KUKA KRL program: MyProgram_244().src

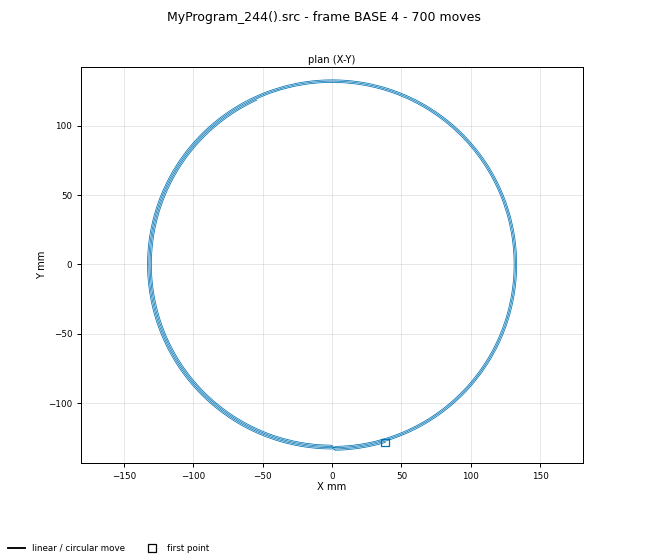
[picture p0: tool path of MyProgram_244().src in frame BASE 4, 700 of 700 moves have a stored position in this frame; points joined in program order, loops and branches not executed]
&ACCESS RVP
&REL 1
&PARAM TEMPLATE = C:\KRC\Roboter\Template\vorgabe
&PARAM EDITMASK = *
DEF MyProgram_244()
; ---- Setting reference (Base) ----
$BASE = BASE_DATA[4]

; --------------------------
; ---- Setting tool (TCP) ----
$TOOL = TOOL_DATA[3]
; --------------------------

$VEL.CP = VEL_APROX_PRINT
Startdeposition()
$VEL.CP = VEL_PRINT
LIN {X 38.4401,Y -128.4466,Z 162,A -74.7058,B 18.9491,C -0.3329,E1 18.9974,E2 523.2154} C_DIS
LIN {X 33.1101,Y -129.9203,Z 162,A -77.04,B 18.9491,C -0.3317,E1 18.9911,E2 525.548} C_DIS
LIN {X 29.9609,Y -130.6824,Z 162,A -78.4866,B 18.9492,C -0.328,E1 18.9871,E2 527.0033} C_DIS
LIN {X 25.973,Y -131.5353,Z 162,A -80.3087,B 18.9492,C -0.3233,E1 18.9821,E2 528.8368} C_DIS
LIN {X 22.2371,Y -132.2161,Z 162,A -81.8211,B 18.9492,C -0.3266,E1 18.978,E2 530.3367} C_DIS
LIN {X 19.1741,Y -132.6951,Z 162,A -83.027,B 18.9492,C -0.3306,E1 18.9747,E2 531.5289} C_DIS
LIN {X 16.3892,Y -133.0686,Z 162,A -84.4176,B 18.9493,C -0.3222,E1 18.9708,E2 532.9437} C_DIS
LIN {X 12.9583,Y -133.4455,Z 162,A -85.833,B 18.9493,C -0.3239,E1 18.9668,E2 534.3526} C_DIS
LIN {X 9.2967,Y -133.7512,Z 162,A -87.5113,B 18.9493,C -0.3189,E1 18.9621,E2 536.0452} C_DIS
LIN {X 5.2547,Y -133.9702,Z 162,A -89.0028,B 18.9493,C -0.3279,E1 18.9581,E2 537.5084} C_DIS
LIN {X 2.1511,Y -134.056,Z 162,A -90.4324,B 18.9493,C -0.3234,E1 18.954,E2 538.9513} C_DIS
LIN {X 2.1511,Y -134.056,Z 162,A -90.4324,B 18.9493,C -0.3234,E1 18.954,E2 538.9513} C_DIS
Enddeposition()
LIN {X 0.9211,Y -133.1439,Z 162,A -90.13,B 17.7288,C -0.2117,E1 17.7322,E2 538.9153} C_DIS
Startdeposition()
$VEL.CP = VEL_PRINT
LIN {X 4.405,Y -133.0795,Z 162,A -88.3392,B 17.7287,C -0.2229,E1 17.7373,E2 537.088} C_DIS
LIN {X 8.2716,Y -132.8933,Z 162,A -86.7196,B 17.7287,C -0.2218,E1 17.7418,E2 535.4731} C_DIS
LIN {X 12.4751,Y -132.5649,Z 162,A -84.9551,B 17.7287,C -0.2207,E1 17.7467,E2 533.7136} C_DIS
LIN {X 16.1435,Y -132.1686,Z 162,A -83.269,B 17.7287,C -0.2253,E1 17.7514,E2 532.0144} C_DIS
LIN {X 20.3858,Y -131.5804,Z 162,A -81.5673,B 17.7287,C -0.221,E1 17.756,E2 530.3288} C_DIS
LIN {X 23.9672,Y -130.9764,Z 162,A -79.9126,B 17.7287,C -0.2256,E1 17.7606,E2 528.6617} C_DIS
LIN {X 28.0553,Y -130.1609,Z 162,A -78.17,B 17.7287,C -0.2251,E1 17.7654,E2 526.924} C_DIS
LIN {X 32.1027,Y -129.2239,Z 162,A -76.0026,B 17.7285,C -0.2413,E1 17.7714,E2 524.7081} C_DIS
LIN {X 35.7552,Y -128.2596,Z 162,A -74.7161,B 17.7286,C -0.2299,E1 17.7747,E2 523.4623} C_DIS
LIN {X 38.9324,Y -127.3311,Z 162,A -72.9424,B 17.7284,C -0.2449,E1 17.7796,E2 521.6439} C_DIS
LIN {X 42.8761,Y -126.0602,Z 162,A -71.6301,B 17.7286,C -0.2287,E1 17.7829,E2 520.3885} C_DIS
LIN {X 46.937,Y -124.603,Z 162,A -69.7312,B 17.7286,C -0.2326,E1 17.7879,E2 518.4825} C_DIS
LIN {X 49.968,Y -123.4186,Z 162,A -68.3823,B 17.7286,C -0.2324,E1 17.7914,E2 517.1386} C_DIS
LIN {X 52.8742,Y -122.2016,Z 162,A -67.036,B 17.7286,C -0.2339,E1 17.7949,E2 515.7921} C_DIS
LIN {X 55.7231,Y -120.9292,Z 162,A -65.1103,B 17.7282,C -0.2587,E1 17.8,E2 513.7926} C_DIS
LIN {X 59.9495,Y -118.8916,Z 162,A -63.7898,B 17.7285,C -0.2344,E1 17.803,E2 512.5568} C_DIS
LIN {X 62.5044,Y -117.5693,Z 162,A -61.9097,B 17.7282,C -0.2615,E1 17.8079,E2 510.5957} C_DIS
LIN {X 66.4149,Y -115.4063,Z 162,A -60.4001,B 17.7284,C -0.2485,E1 17.8114,E2 509.1353} C_DIS
LIN {X 70.1912,Y -113.1488,Z 162,A -58.4889,B 17.7284,C -0.2525,E1 17.816,E2 507.2197} C_DIS
LIN {X 76.278,Y -109.1383,Z 162,A -55.6866,B 17.7284,C -0.2452,E1 17.8224,E2 504.4551} C_DIS
LIN {X 78.609,Y -107.4715,Z 162,A -53.6651,B 17.7279,C -0.2788,E1 17.8272,E2 502.3342} C_DIS
LIN {X 82.5719,Y -104.458,Z 162,A -51.8372,B 17.728,C -0.2706,E1 17.8311,E2 500.5428} C_DIS
LIN {X 85.1779,Y -102.3438,Z 162,A -50.6123,B 17.7281,C -0.265,E1 17.8337,E2 499.3433} C_DIS
LIN {X 88.5691,Y -99.4237,Z 162,A -48.703,B 17.7281,C -0.2685,E1 17.8377,E2 497.4335} C_DIS
LIN {X 92.9776,Y -95.3137,Z 162,A -45.9022,B 17.7279,C -0.2826,E1 17.8434,E2 494.6036} C_DIS
LIN {X 95.4007,Y -92.8885,Z 162,A -44.7083,B 17.7279,C -0.2748,E1 17.8457,E2 493.4425} C_DIS
LIN {X 98.1153,Y -90.0157,Z 162,A -43.0038,B 17.7279,C -0.279,E1 17.8489,E2 491.7353} C_DIS
LIN {X 102.4796,Y -85.0139,Z 162,A -40.1393,B 17.7279,C -0.2863,E1 17.8542,E2 488.8659} C_DIS
LIN {X 107.576,Y -78.4665,Z 162,A -36.8646,B 17.7279,C -0.2835,E1 17.8597,E2 485.6228} C_DIS
LIN {X 112.5667,Y -71.1208,Z 162,A -33.2021,B 17.7278,C -0.2872,E1 17.8654,E2 481.9748} C_DIS
LIN {X 115.0297,Y -67.0654,Z 162,A -30.8023,B 17.7275,C -0.3071,E1 17.8689,E2 479.5279} C_DIS
LIN {X 118.2387,Y -61.2296,Z 162,A -27.4523,B 17.727,C -0.3348,E1 17.8734,E2 476.1134} C_DIS
LIN {X 120.3127,Y -57.043,Z 162,A -26.0674,B 17.7273,C -0.3152,E1 17.875,E2 474.8032} C_DIS
LIN {X 121.6559,Y -54.1186,Z 162,A -24.6633,B 17.7273,C -0.3199,E1 17.8766,E2 473.3947} C_DIS
LIN {X 123.1449,Y -50.6435,Z 162,A -23.0597,B 17.7272,C -0.3237,E1 17.8783,E2 471.7916} C_DIS
LIN {X 125.0396,Y -45.7649,Z 162,A -20.8991,B 17.7272,C -0.3267,E1 17.8805,E2 469.639} C_DIS
LIN {X 126.4553,Y -41.691,Z 162,A -18.9776,B 17.727,C -0.3348,E1 17.8822,E2 467.7065} C_DIS
LIN {X 127.8269,Y -37.2725,Z 162,A -17.0387,B 17.727,C -0.3387,E1 17.8838,E2 465.7711} C_DIS
LIN {X 128.7106,Y -34.0968,Z 162,A -15.5705,B 17.7268,C -0.345,E1 17.8848,E2 464.2947} C_DIS
LIN {X 129.7402,Y -29.942,Z 162,A -13.3916,B 17.7264,C -0.3643,E1 17.8863,E2 462.0712} C_DIS
LIN {X 130.5248,Y -26.3116,Z 162,A -12.4598,B 17.7268,C -0.3422,E1 17.8868,E2 461.2194} C_DIS
LIN {X 130.9612,Y -24.052,Z 162,A -11.1753,B 17.7266,C -0.3571,E1 17.8874,E2 459.8973} C_DIS
LIN {X 131.4541,Y -21.1975,Z 162,A -9.8457,B 17.7264,C -0.3643,E1 17.888,E2 458.5556} C_DIS
LIN {X 132.0314,Y -17.2257,Z 162,A -8.2288,B 17.7264,C -0.3652,E1 17.8887,E2 456.9497} C_DIS
LIN {X 132.4714,Y -13.4488,Z 162,A -6.5412,B 17.7263,C -0.3723,E1 17.8892,E2 455.2535} C_DIS
LIN {X 132.801,Y -9.6401,Z 162,A -5.0073,B 17.7263,C -0.3729,E1 17.8895,E2 453.7309} C_DIS
LIN {X 133.0236,Y -5.8476,Z 162,A -3.2243,B 17.726,C -0.384,E1 17.8897,E2 451.9273} C_DIS
LIN {X 133.1445,Y -1.4544,Z 162,A -1.4344,B 17.726,C -0.3857,E1 17.8898,E2 450.1472} C_DIS
LIN {X 133.1283,Y 2.4386,Z 162,A 0.2134,B 17.7259,C -0.3898,E1 17.8898,E2 448.5003} C_DIS
LIN {X 132.9874,Y 6.5875,Z 162,A 1.9267,B 17.7259,C -0.3923,E1 17.8896,E2 446.7935} C_DIS
LIN {X 132.7248,Y 10.6513,Z 162,A 3.744,B 17.7257,C -0.4003,E1 17.8892,E2 444.9659} C_DIS
LIN {X 132.3728,Y 14.3688,Z 162,A 5.2397,B 17.7257,C -0.4008,E1 17.8888,E2 443.4817} C_DIS
LIN {X 131.8824,Y 18.338,Z 162,A 7.0014,B 17.7255,C -0.4077,E1 17.8882,E2 441.7126} C_DIS
LIN {X 131.2981,Y 22.1322,Z 162,A 8.5557,B 17.7255,C -0.4087,E1 17.8875,E2 440.1681} C_DIS
LIN {X 130.6424,Y 25.7311,Z 162,A 11.1257,B 17.7244,C -0.4538,E1 17.886,E2 437.473} C_DIS
LIN {X 129.1593,Y 32.3575,Z 162,A 12.8777,B 17.7253,C -0.4151,E1 17.885,E2 435.8619} C_DIS
LIN {X 128.1707,Y 36.0732,Z 162,A 14.7264,B 17.7251,C -0.4278,E1 17.8836,E2 433.9874} C_DIS
LIN {X 125.561,Y 44.3161,Z 162,A 18.3458,B 17.7249,C -0.4344,E1 17.8805,E2 430.3762} C_DIS
LIN {X 124.6316,Y 46.8606,Z 162,A 19.568,B 17.7248,C -0.44,E1 17.8793,E2 429.1457} C_DIS
LIN {X 123.1266,Y 50.6874,Z 162,A 21.3856,B 17.7246,C -0.4469,E1 17.8774,E2 427.3203} C_DIS
LIN {X 121.6302,Y 54.176,Z 162,A 22.9095,B 17.7246,C -0.4471,E1 17.8757,E2 425.8079} C_DIS
LIN {X 119.6437,Y 58.432,Z 162,A 25.2502,B 17.7241,C -0.4654,E1 17.8728,E2 423.4259} C_DIS
LIN {X 118.0607,Y 61.5686,Z 162,A 26.232,B 17.7246,C -0.4483,E1 17.8716,E2 422.5074} C_DIS
LIN {X 116.6222,Y 64.2555,Z 162,A 27.8267,B 17.7242,C -0.463,E1 17.8694,E2 420.877} C_DIS
LIN {X 114.3351,Y 68.2415,Z 162,A 29.7403,B 17.7242,C -0.4656,E1 17.8668,E2 418.9691} C_DIS
LIN {X 111.9815,Y 72.0392,Z 162,A 31.6763,B 17.724,C -0.471,E1 17.8639,E2 417.0298} C_DIS
LIN {X 109.5783,Y 75.6449,Z 162,A 33.5648,B 17.7238,C -0.4766,E1 17.8609,E2 415.1367} C_DIS
LIN {X 106.6136,Y 79.7687,Z 162,A 35.6684,B 17.7238,C -0.4786,E1 17.8574,E2 413.0413} C_DIS
LIN {X 104.0275,Y 83.113,Z 162,A 37.4895,B 17.7237,C -0.483,E1 17.8543,E2 411.2185} C_DIS
LIN {X 101.2433,Y 86.4831,Z 162,A 39.3875,B 17.7235,C -0.4879,E1 17.8509,E2 409.3169} C_DIS
LIN {X 98.3103,Y 89.8036,Z 162,A 41.3124,B 17.7235,C -0.4928,E1 17.8473,E2 407.3884} C_DIS
LIN {X 95.1732,Y 93.1209,Z 162,A 43.2319,B 17.7233,C -0.4953,E1 17.8436,E2 405.4731} C_DIS
LIN {X 91.8689,Y 96.3823,Z 162,A 45.2066,B 17.7233,C -0.4985,E1 17.8396,E2 403.4999} C_DIS
LIN {X 88.5887,Y 99.4061,Z 162,A 47.1354,B 17.7231,C -0.5026,E1 17.8356,E2 401.5688} C_DIS
LIN {X 85.7795,Y 101.8399,Z 162,A 48.7338,B 17.7231,C -0.5056,E1 17.8322,E2 399.9698} C_DIS
LIN {X 82.2394,Y 104.7192,Z 162,A 50.6526,B 17.7231,C -0.5075,E1 17.828,E2 398.0553} C_DIS
LIN {X 78.5721,Y 107.4986,Z 162,A 52.6154,B 17.7229,C -0.5103,E1 17.8236,E2 396.0938} C_DIS
LIN {X 74.9854,Y 110.0308,Z 162,A 54.6052,B 17.7227,C -0.5173,E1 17.819,E2 394.091} C_DIS
LIN {X 71.1647,Y 112.5389,Z 162,A 56.4761,B 17.7227,C -0.5166,E1 17.8147,E2 392.231} C_DIS
LIN {X 66.9137,Y 115.1174,Z 162,A 58.7367,B 17.7225,C -0.5244,E1 17.8092,E2 389.9551} C_DIS
LIN {X 63.2973,Y 117.1451,Z 162,A 60.3738,B 17.7226,C -0.5212,E1 17.8052,E2 388.3354} C_DIS
LIN {X 59.7268,Y 119.0044,Z 162,A 61.9869,B 17.7226,C -0.519,E1 17.8013,E2 386.7363} C_DIS
LIN {X 56.9965,Y 120.3349,Z 162,A 63.3153,B 17.7226,C -0.5214,E1 17.7979,E2 385.4051} C_DIS
LIN {X 54.0101,Y 121.7044,Z 162,A 64.8105,B 17.7225,C -0.5261,E1 17.7941,E2 383.8998} C_DIS
LIN {X 49.8646,Y 123.4603,Z 162,A 66.6914,B 17.7225,C -0.5261,E1 17.7892,E2 382.0255} C_DIS
LIN {X 46.3817,Y 124.811,Z 162,A 68.2314,B 17.7225,C -0.5251,E1 17.7852,E2 380.4936} C_DIS
LIN {X 43.3739,Y 125.8876,Z 162,A 69.6353,B 17.7225,C -0.5274,E1 17.7815,E2 379.0862} C_DIS
LIN {X 40.0822,Y 126.9747,Z 162,A 71.3845,B 17.7221,C -0.5383,E1 17.7768,E2 377.306} C_DIS
LIN {X 35.6883,Y 128.2783,Z 162,A 73.0222,B 17.7225,C -0.5272,E1 17.7725,E2 375.7088} C_DIS
LIN {X 32.7382,Y 129.0626,Z 162,A 75.134,B 17.7215,C -0.558,E1 17.7666,E2 373.5005} C_DIS
LIN {X 27.2206,Y 130.3399,Z 162,A 76.7611,B 17.7224,C -0.5289,E1 17.7624,E2 371.972} C_DIS
LIN {X 23.9894,Y 130.9724,Z 162,A 78.318,B 17.7222,C -0.5348,E1 17.758,E2 370.3985} C_DIS
LIN {X 20.4151,Y 131.5759,Z 162,A 79.8044,B 17.7223,C -0.5326,E1 17.754,E2 368.9214} C_DIS
LIN {X 16.969,Y 132.065,Z 162,A 81.3445,B 17.7223,C -0.5346,E1 17.7497,E2 367.3765} C_DIS
LIN {X 12.8514,Y 132.5288,Z 162,A 83.0922,B 17.7223,C -0.5337,E1 17.7449,E2 365.6337} C_DIS
LIN {X 8.8949,Y 132.8549,Z 162,A 84.9027,B 17.7222,C -0.5376,E1 17.7398,E2 363.8117} C_DIS
LIN {X 4.989,Y 133.0571,Z 162,A 86.4461,B 17.7223,C -0.5325,E1 17.7355,E2 362.2857} C_DIS
LIN {X 0.9974,Y 133.147,Z 162,A 88.2211,B 17.7223,C -0.5345,E1 17.7305,E2 360.5046} C_DIS
LIN {X -2.4674,Y 133.1279,Z 162,A 89.7391,B 17.7223,C -0.5352,E1 17.7263,E2 358.9841} C_DIS
LIN {X -6.5137,Y 132.9911,Z 162,A 91.4349,B 17.7223,C -0.5331,E1 17.7216,E2 357.2948} C_DIS
LIN {X -9.9735,Y 132.7766,Z 162,A 92.9352,B 17.7223,C -0.5329,E1 17.7174,E2 355.7943} C_DIS
LIN {X -14.1183,Y 132.3998,Z 162,A 94.7247,B 17.7223,C -0.5321,E1 17.7124,E2 354.0061} C_DIS
LIN {X -17.8365,Y 131.9513,Z 162,A 96.4127,B 17.7223,C -0.534,E1 17.7077,E2 352.3101} C_DIS
LIN {X -21.7102,Y 131.3685,Z 162,A 98.327,B 17.722,C -0.5413,E1 17.7024,E2 350.3695} C_DIS
LIN {X -24.9922,Y 130.7837,Z 162,A 99.4282,B 17.7224,C -0.5283,E1 17.6995,E2 349.3093} C_DIS
LIN {X -31.9254,Y 129.2683,Z 162,A 102.4778,B 17.7225,C -0.5256,E1 17.6912,E2 346.2628} C_DIS
LIN {X -34.6255,Y 128.5696,Z 162,A 103.794,B 17.7225,C -0.5287,E1 17.6876,E2 344.9337} C_DIS
LIN {X -43.6563,Y 125.7897,Z 162,A 107.4467,B 17.723,C -0.5097,E1 17.678,E2 341.334} C_DIS
LIN {X -46.9349,Y 124.6038,Z 162,A 109.308,B 17.7226,C -0.5207,E1 17.673,E2 339.4312} C_DIS
LIN {X -50.5818,Y 123.1707,Z 162,A 111.3581,B 17.7223,C -0.5314,E1 17.6676,E2 337.3393} C_DIS
LIN {X -53.8283,Y 121.7857,Z 162,A 112.4133,B 17.7229,C -0.513,E1 17.6651,E2 336.3411} C_DIS
LIN {X -56.6826,Y 120.4849,Z 162,A 114.1908,B 17.7225,C -0.5261,E1 17.6604,E2 334.5138} C_DIS
LIN {X -59.6374,Y 119.0489,Z 162,A 115.973,B 17.7222,C -0.537,E1 17.6559,E2 332.6888} C_DIS
LIN {X -64.3129,Y 116.5904,Z 162,A 117.425,B 17.7231,C -0.5046,E1 17.6526,E2 331.3378} C_DIS
LIN {X -66.9437,Y 115.1001,Z 162,A 118.9992,B 17.7229,C -0.512,E1 17.6487,E2 329.7325} C_DIS
LIN {X -70.7861,Y 112.7779,Z 162,A 121.021,B 17.7229,C -0.5117,E1 17.6438,E2 327.7021} C_DIS
LIN {X -74.994,Y 110.025,Z 162,A 123.0696,B 17.7231,C -0.5038,E1 17.6391,E2 325.6699} C_DIS
LIN {X -79.5511,Y 106.7756,Z 162,A 125.2577,B 17.7234,C -0.4916,E1 17.6343,E2 323.5109} C_DIS
LIN {X -82.004,Y 104.904,Z 162,A 126.8766,B 17.7232,C -0.499,E1 17.6306,E2 321.859} C_DIS
LIN {X -85.898,Y 101.739,Z 162,A 129.4235,B 17.723,C -0.5079,E1 17.625,E2 319.2684} C_DIS
LIN {X -89.1638,Y 98.8909,Z 162,A 130.7262,B 17.7236,C -0.4845,E1 17.6225,E2 318.0354} C_DIS
LIN {X -91.6865,Y 96.5567,Z 162,A 132.9844,B 17.723,C -0.5081,E1 17.6177,E2 315.6857} C_DIS
LIN {X -95.4305,Y 92.8577,Z 162,A 135.1689,B 17.7232,C -0.5001,E1 17.6135,E2 313.5139} C_DIS
LIN {X -98.6883,Y 89.3871,Z 162,A 136.5035,B 17.724,C -0.4708,E1 17.6111,E2 312.2677} C_DIS
LIN {X -100.9612,Y 86.8116,Z 162,A 138.3748,B 17.7237,C -0.4807,E1 17.6076,E2 310.3515} C_DIS
LIN {X -104.1069,Y 83.0131,Z 162,A 140.3623,B 17.724,C -0.4708,E1 17.6042,E2 308.3832} C_DIS
LIN {X -106.758,Y 79.5748,Z 162,A 142.2426,B 17.7241,C -0.4665,E1 17.601,E2 306.504} C_DIS
LIN {X -109.469,Y 75.8026,Z 162,A 144.4981,B 17.7241,C -0.47,E1 17.5973,E2 304.2206} C_DIS
LIN {X -111.4017,Y 72.9328,Z 162,A 145.6418,B 17.7244,C -0.4543,E1 17.5956,E2 303.1204} C_DIS
LIN {X -114.2198,Y 68.4351,Z 162,A 147.7787,B 17.7247,C -0.4432,E1 17.5925,E2 301.0043} C_DIS
LIN {X -115.7253,Y 65.8566,Z 162,A 149.3559,B 17.7245,C -0.4495,E1 17.5903,E2 299.3942} C_DIS
LIN {X -117.7258,Y 62.2065,Z 162,A 151.5968,B 17.7243,C -0.4598,E1 17.5873,E2 297.1018} C_DIS
LIN {X -119.7405,Y 58.234,Z 162,A 153.2256,B 17.7246,C -0.4446,E1 17.5853,E2 295.5106} C_DIS
LIN {X -121.8148,Y 53.7632,Z 162,A 155.3479,B 17.7248,C -0.4386,E1 17.5829,E2 293.3912} C_DIS
LIN {X -124.1451,Y 48.1345,Z 162,A 157.7942,B 17.7251,C -0.425,E1 17.5804,E2 290.9698} C_DIS
LIN {X -125.3038,Y 45.0323,Z 162,A 159.2043,B 17.7252,C -0.4203,E1 17.579,E2 289.5636} C_DIS
LIN {X -126.5386,Y 41.4408,Z 162,A 161.1164,B 17.7252,C -0.4248,E1 17.5773,E2 287.6207} C_DIS
LIN {X -128.4223,Y 35.1736,Z 162,A 163.6718,B 17.7255,C -0.4076,E1 17.5753,E2 285.1008} C_DIS
LIN {X -129.1451,Y 32.4134,Z 162,A 164.9402,B 17.7255,C -0.4053,E1 17.5744,E2 283.8293} C_DIS
LIN {X -130.6342,Y 25.7741,Z 162,A 168.2618,B 17.7255,C -0.4095,E1 17.5725,E2 280.4649} C_DIS
LIN {X -131.2524,Y 22.4034,Z 162,A 169.5416,B 17.7257,C -0.3985,E1 17.5719,E2 279.2107} C_DIS
LIN {X -131.8734,Y 18.4007,Z 162,A 171.7432,B 17.7255,C -0.4086,E1 17.571,E2 276.9563} C_DIS
LIN {X -132.4547,Y 13.6075,Z 162,A 173.4419,B 17.7259,C -0.3894,E1 17.5705,E2 275.3064} C_DIS
LIN {X -132.7637,Y 10.1499,Z 162,A 174.8116,B 17.7261,C -0.3806,E1 17.5702,E2 273.9538} C_DIS
LIN {X -133.0072,Y 6.1945,Z 162,A 176.5855,B 17.7261,C -0.3776,E1 17.57,E2 272.1741} C_DIS
LIN {X -133.1499,Y 0.6535,Z 162,A 179.0729,B 17.7262,C -0.3737,E1 17.5698,E2 269.6778} C_DIS
LIN {X -133.0912,Y -3.9837,Z 162,A -179.0232,B 17.7264,C -0.3644,E1 17.57,E2 267.7877} C_DIS
LIN {X -132.9015,Y -8.1385,Z 162,A -177.2896,B 17.7266,C -0.3571,E1 17.5702,E2 266.0633} C_DIS
LIN {X -132.51,Y -13.0469,Z 162,A -175.2686,B 17.7268,C -0.3473,E1 17.5707,E2 264.057} C_DIS
LIN {X -131.6927,Y -19.6607,Z 162,A -172.319,B 17.7268,C -0.3412,E1 17.5718,E2 261.1016} C_DIS
LIN {X -131.0164,Y -23.7438,Z 162,A -170.2086,B 17.7268,C -0.347,E1 17.5728,E2 258.9537} C_DIS
LIN {X -130.3,Y -27.4114,Z 162,A -168.7136,B 17.7269,C -0.3383,E1 17.5736,E2 257.4746} C_DIS
LIN {X -129.2408,Y -32.0364,Z 162,A -166.8324,B 17.7271,C -0.3269,E1 17.5748,E2 255.6153} C_DIS
LIN {X -128.2073,Y -35.9422,Z 162,A -165.0386,B 17.7271,C -0.3236,E1 17.5761,E2 253.8169} C_DIS
LIN {X -127.2376,Y -39.2379,Z 162,A -163.5455,B 17.7273,C -0.3198,E1 17.5773,E2 252.3239} C_DIS
LIN {X -126.252,Y -42.3016,Z 162,A -162.1634,B 17.7273,C -0.3157,E1 17.5785,E2 250.9438} C_DIS
LIN {X -125.0828,Y -45.6452,Z 162,A -160.6097,B 17.7273,C -0.3124,E1 17.58,E2 249.3883} C_DIS
LIN {X -123.4363,Y -49.924,Z 162,A -158.6021,B 17.7275,C -0.308,E1 17.582,E2 247.3787} C_DIS
LIN {X -122.0265,Y -53.2791,Z 162,A -156.9886,B 17.7275,C -0.3053,E1 17.5838,E2 245.7612} C_DIS
LIN {X -118.9985,Y -59.7395,Z 162,A -153.9874,B 17.7277,C -0.2945,E1 17.5874,E2 242.7717} C_DIS
LIN {X -117.7216,Y -62.2144,Z 162,A -152.7089,B 17.7277,C -0.2941,E1 17.5891,E2 241.4847} C_DIS
LIN {X -115.6817,Y -65.933,Z 162,A -150.8034,B 17.7277,C -0.2921,E1 17.5917,E2 239.5714} C_DIS
LIN {X -113.3681,Y -69.8366,Z 162,A -148.659,B 17.7277,C -0.2937,E1 17.5948,E2 237.4056} C_DIS
LIN {X -110.985,Y -73.5658,Z 162,A -147.1433,B 17.728,C -0.2755,E1 17.5971,E2 235.9388} C_DIS
LIN {X -109.1237,Y -76.299,Z 162,A -145.5502,B 17.728,C -0.2779,E1 17.5996,E2 234.3263} C_DIS
LIN {X -106.6318,Y -79.7443,Z 162,A -143.6861,B 17.728,C -0.2747,E1 17.6027,E2 232.4596} C_DIS
LIN {X -103.9378,Y -83.2256,Z 162,A -141.8161,B 17.728,C -0.2695,E1 17.6059,E2 230.5941} C_DIS
LIN {X -101.4436,Y -86.2474,Z 162,A -139.679,B 17.7279,C -0.2814,E1 17.6099,E2 228.4032} C_DIS
LIN {X -98.758,Y -89.3102,Z 162,A -138.6032,B 17.7283,C -0.2539,E1 17.6117,E2 227.4112} C_DIS
LIN {X -96.7778,Y -91.4521,Z 162,A -137.0477,B 17.7282,C -0.2617,E1 17.6148,E2 225.8202} C_DIS
LIN {X -93.7145,Y -94.5888,Z 162,A -135.119,B 17.7282,C -0.2592,E1 17.6186,E2 223.8876} C_DIS
LIN {X -90.3961,Y -97.7656,Z 162,A -133.3724,B 17.7284,C -0.2472,E1 17.622,E2 222.1702} C_DIS
LIN {X -88.1061,Y -99.8336,Z 162,A -131.8304,B 17.7284,C -0.2522,E1 17.6253,E2 220.6029} C_DIS
LIN {X -83.005,Y -104.1134,Z 162,A -129.1857,B 17.7284,C -0.2391,E1 17.631,E2 217.9866} C_DIS
LIN {X -80.5913,Y -105.9934,Z 162,A -127.5502,B 17.7284,C -0.2481,E1 17.6346,E2 216.313} C_DIS
LIN {X -77.769,Y -108.0813,Z 162,A -125.9641,B 17.7284,C -0.2482,E1 17.6382,E2 214.7183} C_DIS
LIN {X -74.2414,Y -110.534,Z 162,A -124.1683,B 17.7284,C -0.2434,E1 17.6424,E2 212.9297} C_DIS
LIN {X -70.2026,Y -113.1414,Z 162,A -121.9915,B 17.7284,C -0.2441,E1 17.6475,E2 210.7404} C_DIS
LIN {X -67.1395,Y -114.9862,Z 162,A -120.5861,B 17.7285,C -0.2371,E1 17.6509,E2 209.3518} C_DIS
LIN {X -63.395,Y -117.0925,Z 162,A -118.7317,B 17.7285,C -0.2349,E1 17.6554,E2 207.4972} C_DIS
LIN {X -60.2441,Y -118.7416,Z 162,A -117.2429,B 17.7285,C -0.2315,E1 17.6591,E2 206.0137} C_DIS
LIN {X -57.0225,Y -120.3225,Z 162,A -115.621,B 17.7285,C -0.2324,E1 17.6632,E2 204.3825} C_DIS
LIN {X -52.9041,Y -122.1887,Z 162,A -113.7705,B 17.7286,C -0.2269,E1 17.6679,E2 202.5438} C_DIS
LIN {X -49.376,Y -123.6572,Z 162,A -112.1541,B 17.7286,C -0.2242,E1 17.6721,E2 200.931} C_DIS
LIN {X -46.0174,Y -124.9474,Z 162,A -110.4396,B 17.7286,C -0.2288,E1 17.6766,E2 199.1963} C_DIS
LIN {X -41.7412,Y -126.4386,Z 162,A -108.6802,B 17.7287,C -0.2203,E1 17.6812,E2 197.4601} C_DIS
LIN {X -38.8691,Y -127.3505,Z 162,A -107.3289,B 17.7287,C -0.2213,E1 17.6848,E2 196.1019} C_DIS
LIN {X -35.3736,Y -128.3663,Z 162,A -105.1264,B 17.7284,C -0.2437,E1 17.691,E2 193.8209} C_DIS
LIN {X -30.4385,Y -129.6267,Z 162,A -103.4581,B 17.7287,C -0.2231,E1 17.6953,E2 192.217} C_DIS
LIN {X -26.5938,Y -130.4674,Z 162,A -101.8796,B 17.7287,C -0.2181,E1 17.6996,E2 190.6523} C_DIS
LIN {X -23.3024,Y -131.0954,Z 162,A -100.4365,B 17.7287,C -0.2176,E1 17.7036,E2 189.2087} C_DIS
LIN {X -19.6947,Y -131.6874,Z 162,A -98.7223,B 17.7287,C -0.2223,E1 17.7083,E2 187.4768} C_DIS
LIN {X -15.6772,Y -132.2242,Z 162,A -97.0825,B 17.7287,C -0.2181,E1 17.7128,E2 185.8492} C_DIS
LIN {X -11.4328,Y -132.6588,Z 162,A -95.2758,B 17.7287,C -0.2168,E1 17.7179,E2 184.0454} C_DIS
LIN {X -7.9397,Y -132.9137,Z 162,A -93.7673,B 17.7287,C -0.2168,E1 17.7221,E2 182.5362} C_DIS
LIN {X -3.9265,Y -133.0927,Z 162,A -92.0182,B 17.7287,C -0.2176,E1 17.727,E2 180.7838} C_DIS
LIN {X 0.0972,Y -133.152,Z 162,A -90.1654,B 17.7287,C -0.2224,E1 17.7322,E2 178.9153} C_DIS
LIN {X 0.0972,Y -133.152,Z 162,A -90.1654,B 17.7287,C -0.2224,E1 17.7322,E2 178.9153} C_DIS
Enddeposition()
LIN {X 0.913,Y -132.2218,Z 162,A -89.6358,B 15.9112,C -0.0387,E1 15.9133,E2 178.9141} C_DIS
Startdeposition()
$VEL.CP = VEL_PRINT
LIN {X -2.0763,Y -132.2115,Z 162,A -91.3724,B 15.9112,C -0.0239,E1 15.9083,E2 180.7047} C_DIS
LIN {X -5.8273,Y -132.1009,Z 162,A -93.1059,B 15.9112,C -0.0203,E1 15.9034,E2 182.452} C_DIS
LIN {X -9.6628,Y -131.8741,Z 162,A -94.6183,B 15.9112,C -0.0253,E1 15.8993,E2 183.9466} C_DIS
LIN {X -13.0166,Y -131.5859,Z 162,A -96.2011,B 15.9112,C -0.0215,E1 15.8948,E2 185.5449} C_DIS
LIN {X -17.2208,Y -131.1014,Z 162,A -97.9455,B 15.9112,C -0.0248,E1 15.89,E2 187.2792} C_DIS
LIN {X -20.7076,Y -130.5969,Z 162,A -99.4487,B 15.9112,C -0.026,E1 15.8859,E2 188.78} C_DIS
LIN {X -24.3758,Y -129.962,Z 162,A -101.1338,B 15.9112,C -0.0242,E1 15.8812,E2 190.4742} C_DIS
LIN {X -27.9059,Y -129.2492,Z 162,A -102.6631,B 15.9112,C -0.026,E1 15.8771,E2 192} C_DIS
LIN {X -33.4122,Y -127.9377,Z 162,A -105.3248,B 15.9112,C -0.0207,E1 15.8698,E2 194.6871} C_DIS
LIN {X -38.4693,Y -126.5078,Z 162,A -107.6091,B 15.9112,C -0.0221,E1 15.8636,E2 196.9726} C_DIS
LIN {X -43.639,Y -124.8191,Z 162,A -109.7377,B 15.9112,C -0.0312,E1 15.8581,E2 199.074} C_DIS
LIN {X -46.6682,Y -123.7183,Z 162,A -111.1326,B 15.9112,C -0.0326,E1 15.8544,E2 200.4686} C_DIS
LIN {X -49.5915,Y -122.5755,Z 162,A -112.5187,B 15.9112,C -0.0331,E1 15.8508,E2 201.8578} C_DIS
LIN {X -52.691,Y -121.2755,Z 162,A -113.9779,B 15.9112,C -0.0345,E1 15.8471,E2 203.3173} C_DIS
LIN {X -55.7441,Y -119.9028,Z 162,A -115.4326,B 15.9112,C -0.036,E1 15.8434,E2 204.7724} C_DIS
LIN {X -58.9056,Y -118.3822,Z 162,A -116.9608,B 15.9112,C -0.0376,E1 15.8395,E2 206.3013} C_DIS
LIN {X -62.4922,Y -116.5301,Z 162,A -118.8164,B 15.9112,C -0.0364,E1 15.8349,E2 208.1693} C_DIS
LIN {X -66.1324,Y -114.5036,Z 162,A -120.6196,B 15.9112,C -0.039,E1 15.8306,E2 209.9719} C_DIS
LIN {X -70.7202,Y -111.7284,Z 162,A -122.8999,B 15.9112,C -0.0437,E1 15.8251,E2 212.2465} C_DIS
LIN {X -74.235,Y -109.4245,Z 162,A -124.9956,B 15.9112,C -0.038,E1 15.8202,E2 214.3743} C_DIS
LIN {X -76.8944,Y -107.5722,Z 162,A -126.3182,B 15.9112,C -0.0428,E1 15.8172,E2 215.6867} C_DIS
LIN {X -79.9442,Y -105.3262,Z 162,A -127.8486,B 15.9112,C -0.049,E1 15.8138,E2 217.2034} C_DIS
LIN {X -83.9586,Y -102.1547,Z 162,A -130.4268,B 15.9112,C -0.0419,E1 15.8081,E2 219.8233} C_DIS
LIN {X -86.9606,Y -99.6112,Z 162,A -131.7286,B 15.9112,C -0.0575,E1 15.8055,E2 221.0765} C_DIS
LIN {X -90.0605,Y -96.8176,Z 162,A -133.4695,B 15.9112,C -0.063,E1 15.8019,E2 222.8085} C_DIS
LIN {X -92.7124,Y -94.2813,Z 162,A -135.2026,B 15.9112,C -0.0618,E1 15.7984,E2 224.5577} C_DIS
LIN {X -95.6764,Y -91.272,Z 162,A -137.0513,B 15.9112,C -0.0651,E1 15.7948,E2 226.4076} C_DIS
LIN {X -99.4106,Y -87.1897,Z 162,A -139.6603,B 15.9112,C -0.0639,E1 15.7899,E2 229.0401} C_DIS
LIN {X -102.8714,Y -83.0784,Z 162,A -141.6715,B 15.9111,C -0.0787,E1 15.7864,E2 231.0121} C_DIS
LIN {X -105.1059,Y -80.2329,Z 162,A -143.3724,B 15.9111,C -0.0783,E1 15.7835,E2 232.7277} C_DIS
LIN {X -107.7509,Y -76.6445,Z 162,A -145.3717,B 15.9111,C -0.0808,E1 15.7802,E2 234.7334} C_DIS
LIN {X -109.6721,Y -73.8692,Z 162,A -146.8157,B 15.9111,C -0.0849,E1 15.7779,E2 236.1741} C_DIS
LIN {X -112.4013,Y -69.646,Z 162,A -148.7652,B 15.911,C -0.0972,E1 15.775,E2 238.0946} C_DIS
LIN {X -114.1027,Y -66.8218,Z 162,A -150.4555,B 15.911,C -0.093,E1 15.7726,E2 239.8146} C_DIS
LIN {X -116.2747,Y -62.9675,Z 162,A -152.4156,B 15.911,C -0.0967,E1 15.7699,E2 241.7781} C_DIS
LIN {X -118.1528,Y -59.3668,Z 162,A -154.3956,B 15.911,C -0.0948,E1 15.7674,E2 243.7823} C_DIS
LIN {X -119.593,Y -56.4074,Z 162,A -155.9396,B 15.911,C -0.0952,E1 15.7655,E2 245.3388} C_DIS
LIN {X -121.1951,Y -52.877,Z 162,A -157.1568,B 15.9109,C -0.1134,E1 15.7642,E2 246.4999} C_DIS
LIN {X -122.6959,Y -49.2926,Z 162,A -158.8633,B 15.9109,C -0.1174,E1 15.7624,E2 248.2074} C_DIS
LIN {X -123.9386,Y -46.08,Z 162,A -160.3953,B 15.9109,C -0.1204,E1 15.7609,E2 249.7424} C_DIS
LIN {X -125.0742,Y -42.9031,Z 162,A -162.0288,B 15.9109,C -0.1195,E1 15.7594,E2 251.3946} C_DIS
LIN {X -126.389,Y -38.8576,Z 162,A -163.7609,B 15.9108,C -0.128,E1 15.7579,E2 253.1117} C_DIS
LIN {X -127.3882,Y -35.4448,Z 162,A -165.271,B 15.9108,C -0.1334,E1 15.7567,E2 254.6164} C_DIS
LIN {X -128.36,Y -31.7555,Z 162,A -167.2224,B 15.9108,C -0.1294,E1 15.7554,E2 256.601} C_DIS
LIN {X -129.4982,Y -26.7294,Z 162,A -169.7185,B 15.9108,C -0.1283,E1 15.7539,E2 259.1252} C_DIS
LIN {X -130.3024,Y -22.4932,Z 162,A -171.0705,B 15.9106,C -0.1489,E1 15.7533,E2 260.4145} C_DIS
LIN {X -130.9834,Y -18.1061,Z 162,A -173.5388,B 15.9106,C -0.1388,E1 15.7523,E2 262.9443} C_DIS
LIN {X -131.4787,Y -14.0534,Z 162,A -174.4726,B 15.9104,C -0.1685,E1 15.752,E2 263.7779} C_DIS
LIN {X -131.9362,Y -8.8001,Z 162,A -177.0797,B 15.9104,C -0.1659,E1 15.7514,E2 266.4203} C_DIS
LIN {X -132.0977,Y -5.9058,Z 162,A -178.5518,B 15.9104,C -0.1634,E1 15.7512,E2 267.9162} C_DIS
LIN {X -132.2298,Y 0.2327,Z 162,A 178.3466,B 15.9105,C -0.1587,E1 15.7511,E2 271.0657} C_DIS
LIN {X -132.147,Y 4.647,Z 162,A 177.0959,B 15.9102,C -0.1837,E1 15.7512,E2 272.2366} C_DIS
LIN {X -131.941,Y 8.7218,Z 162,A 174.6916,B 15.9104,C -0.1706,E1 15.7516,E2 274.7128} C_DIS
LIN {X -131.607,Y 12.7973,Z 162,A 173.177,B 15.9102,C -0.1835,E1 15.752,E2 276.1952} C_DIS
LIN {X -131.0901,Y 17.3071,Z 162,A 171.3589,B 15.9102,C -0.1937,E1 15.7526,E2 277.9932} C_DIS
LIN {X -129.97,Y 24.3339,Z 162,A 168.2605,B 15.91,C -0.2026,E1 15.754,E2 281.0893} C_DIS
LIN {X -128.8971,Y 29.4896,Z 162,A 166.0328,B 15.91,C -0.211,E1 15.7553,E2 283.3075} C_DIS
LIN {X -128.1583,Y 32.5505,Z 162,A 164.5646,B 15.9099,C -0.212,E1 15.7563,E2 284.786} C_DIS
LIN {X -127.1252,Y 36.3849,Z 162,A 162.3541,B 15.91,C -0.2029,E1 15.758,E2 287.051} C_DIS
LIN {X -125.9132,Y 40.3726,Z 162,A 161.0336,B 15.9098,C -0.2223,E1 15.7591,E2 288.3127} C_DIS
LIN {X -124.7035,Y 43.9723,Z 162,A 159.2499,B 15.9098,C -0.2231,E1 15.7607,E2 290.1102} C_DIS
LIN {X -123.0698,Y 48.3537,Z 162,A 157.3306,B 15.9096,C -0.232,E1 15.7626,E2 292.0142} C_DIS
LIN {X -121.9272,Y 51.1648,Z 162,A 156.024,B 15.9096,C -0.236,E1 15.764,E2 293.3181} C_DIS
LIN {X -120.5646,Y 54.2984,Z 162,A 154.5164,B 15.9096,C -0.2394,E1 15.7657,E2 294.8268} C_DIS
LIN {X -119.023,Y 57.602,Z 162,A 152.2764,B 15.9097,C -0.2246,E1 15.7685,E2 297.1412} C_DIS
LIN {X -116.7735,Y 62.0352,Z 162,A 150.8412,B 15.9093,C -0.2515,E1 15.7703,E2 298.4901} C_DIS
LIN {X -115.0565,Y 65.1668,Z 162,A 149.0832,B 15.9093,C -0.2495,E1 15.7727,E2 300.2706} C_DIS
LIN {X -111.925,Y 70.4086,Z 162,A 146.5961,B 15.9092,C -0.2612,E1 15.7763,E2 302.7357} C_DIS
LIN {X -109.2271,Y 74.5259,Z 162,A 144.4674,B 15.9091,C -0.2668,E1 15.7795,E2 304.861} C_DIS
LIN {X -107.4,Y 77.1353,Z 162,A 142.9333,B 15.9091,C -0.2658,E1 15.782,E2 306.4112} C_DIS
LIN {X -104.9735,Y 80.4059,Z 162,A 141.1015,B 15.9091,C -0.2682,E1 15.7851,E2 308.2485} C_DIS
LIN {X -101.5497,Y 84.6898,Z 162,A 138.6963,B 15.909,C -0.2731,E1 15.7894,E2 310.654} C_DIS
LIN {X -98.7213,Y 87.9702,Z 162,A 136.808,B 15.909,C -0.2772,E1 15.7928,E2 312.5411} C_DIS
LIN {X -94.9122,Y 92.0665,Z 162,A 134.0546,B 15.909,C -0.273,E1 15.7982,E2 315.3296} C_DIS
LIN {X -92.2155,Y 94.7678,Z 162,A 132.6871,B 15.9088,C -0.2851,E1 15.8008,E2 316.6619} C_DIS
LIN {X -89.0885,Y 97.7132,Z 162,A 130.8502,B 15.9088,C -0.2898,E1 15.8046,E2 318.4937} C_DIS
LIN {X -82.9246,Y 102.9954,Z 162,A 127.3002,B 15.9086,C -0.296,E1 15.8122,E2 322.0433} C_DIS
LIN {X -79.3469,Y 105.7769,Z 162,A 125.1329,B 15.9086,C -0.2937,E1 15.817,E2 324.232} C_DIS
LIN {X -74.8517,Y 109.0035,Z 162,A 123.1315,B 15.9083,C -0.3101,E1 15.8215,E2 326.1845} C_DIS
LIN {X -72.1288,Y 110.8242,Z 162,A 121.4709,B 15.9084,C -0.3053,E1 15.8254,E2 327.8717} C_DIS
LIN {X -68.2617,Y 113.2472,Z 162,A 119.5195,B 15.9084,C -0.3094,E1 15.83,E2 329.8179} C_DIS
LIN {X -64.491,Y 115.4364,Z 162,A 116.3564,B 15.909,C -0.274,E1 15.8382,E2 333.1254} C_DIS
LIN {X -57.0382,Y 119.2924,Z 162,A 114.3384,B 15.908,C -0.3283,E1 15.8427,E2 334.9533} C_DIS
LIN {X -51.5571,Y 121.7634,Z 162,A 111.485,B 15.908,C -0.3241,E1 15.85,E2 337.8333} C_DIS
LIN {X -47.7364,Y 123.3098,Z 162,A 109.6097,B 15.908,C -0.3235,E1 15.8549,E2 339.7174} C_DIS
LIN {X -44.259,Y 124.6017,Z 162,A 107.9618,B 15.908,C -0.3241,E1 15.8592,E2 341.3686} C_DIS
LIN {X -35.2355,Y 127.4468,Z 162,A 103.783,B 15.908,C -0.3257,E1 15.8704,E2 345.5532} C_DIS
LIN {X -26.8867,Y 129.4661,Z 162,A 100.2782,B 15.9078,C -0.3354,E1 15.8799,E2 349.03} C_DIS
LIN {X -23.3798,Y 130.1441,Z 162,A 98.5899,B 15.9078,C -0.332,E1 15.8845,E2 350.7336} C_DIS
LIN {X -20.4499,Y 130.6368,Z 162,A 97.2983,B 15.9078,C -0.3327,E1 15.8881,E2 352.0248} C_DIS
LIN {X -16.9587,Y 131.1357,Z 162,A 95.7945,B 15.9078,C -0.3342,E1 15.8923,E2 353.5247} C_DIS
LIN {X -13.0661,Y 131.5812,Z 162,A 94.0105,B 15.9078,C -0.3322,E1 15.8972,E2 355.3178} C_DIS
LIN {X -9.2969,Y 131.9008,Z 162,A 92.4471,B 15.9078,C -0.3352,E1 15.9016,E2 356.8714} C_DIS
LIN {X -5.4257,Y 132.1166,Z 162,A 90.7231,B 15.9078,C -0.3342,E1 15.9064,E2 358.5997} C_DIS
LIN {X -1.7646,Y 132.2167,Z 162,A 89.0941,B 15.9078,C -0.3331,E1 15.9109,E2 360.2328} C_DIS
LIN {X 2.3254,Y 132.2073,Z 162,A 87.4052,B 15.9078,C -0.3359,E1 15.9156,E2 361.9111} C_DIS
LIN {X 5.8387,Y 132.1005,Z 162,A 85.7174,B 15.9079,C -0.3306,E1 15.9204,E2 363.6175} C_DIS
LIN {X 9.9076,Y 131.8562,Z 162,A 84.0074,B 15.9079,C -0.3322,E1 15.9251,E2 365.3203} C_DIS
LIN {X 14.1565,Y 131.4676,Z 162,A 82.2564,B 15.9079,C -0.335,E1 15.93,E2 367.0592} C_DIS
LIN {X 17.7841,Y 131.0275,Z 162,A 80.5546,B 15.9079,C -0.3307,E1 15.9347,E2 368.7744} C_DIS
LIN {X 22.0391,Y 130.3782,Z 162,A 78.7895,B 15.9079,C -0.3333,E1 15.9395,E2 370.5272} C_DIS
LIN {X 26.2204,Y 129.6017,Z 162,A 76.0227,B 15.9085,C -0.3024,E1 15.9474,E2 373.4009} C_DIS
LIN {X 32.6828,Y 128.1247,Z 162,A 74.5014,B 15.9076,C -0.3448,E1 15.9511,E2 374.7644} C_DIS
LIN {X 38.1527,Y 126.6047,Z 162,A 71.7656,B 15.9079,C -0.3338,E1 15.9586,E2 377.5326} C_DIS
LIN {X 41.7985,Y 125.447,Z 162,A 70.0159,B 15.9079,C -0.3294,E1 15.9632,E2 379.293} C_DIS
LIN {X 45.0514,Y 124.316,Z 162,A 68.525,B 15.9079,C -0.3281,E1 15.9672,E2 380.7837} C_DIS
LIN {X 48.0968,Y 123.1697,Z 162,A 67.112,B 15.908,C -0.3266,E1 15.9708,E2 382.1971} C_DIS
LIN {X 51.0935,Y 121.957,Z 162,A 65.7074,B 15.908,C -0.325,E1 15.9745,E2 383.6022} C_DIS
LIN {X 54.3157,Y 120.5569,Z 162,A 64.1754,B 15.908,C -0.3229,E1 15.9784,E2 385.1355} C_DIS
LIN {X 57.9441,Y 118.8565,Z 162,A 62.5581,B 15.908,C -0.3248,E1 15.9824,E2 386.739} C_DIS
LIN {X 61.0589,Y 117.2861,Z 162,A 60.9327,B 15.9082,C -0.319,E1 15.9865,E2 388.3781} C_DIS
LIN {X 64.7693,Y 115.28,Z 162,A 58.8139,B 15.9084,C -0.3067,E1 15.9918,E2 390.5315} C_DIS
LIN {X 67.7178,Y 113.5731,Z 162,A 57.712,B 15.9082,C -0.3172,E1 15.9943,E2 391.5898} C_DIS
LIN {X 70.9886,Y 111.5585,Z 162,A 55.8848,B 15.9083,C -0.3091,E1 15.9987,E2 393.4366} C_DIS
LIN {X 74.9272,Y 108.9517,Z 162,A 53.8665,B 15.9083,C -0.3068,E1 16.0034,E2 395.4522} C_DIS
LIN {X 78.0921,Y 106.7062,Z 162,A 52.194,B 15.9084,C -0.3043,E1 16.0071,E2 397.1243} C_DIS
LIN {X 81.8196,Y 103.8755,Z 162,A 50.2096,B 15.9084,C -0.3022,E1 16.0115,E2 399.1044} C_DIS
LIN {X 84.151,Y 101.9961,Z 162,A 48.9192,B 15.9085,C -0.3,E1 16.0143,E2 400.3945} C_DIS
LIN {X 87.3658,Y 99.2564,Z 162,A 47.06,B 15.9086,C -0.2955,E1 16.0182,E2 402.2581} C_DIS
LIN {X 90.7509,Y 96.1708,Z 162,A 45.1144,B 15.9086,C -0.2929,E1 16.0222,E2 404.2} C_DIS
LIN {X 93.995,Y 93.0029,Z 162,A 43.18,B 15.9087,C -0.2899,E1 16.026,E2 406.132} C_DIS
LIN {X 97.028,Y 89.8346,Z 162,A 41.2657,B 15.9087,C -0.2854,E1 16.0297,E2 408.0491} C_DIS
LIN {X 99.9652,Y 86.5541,Z 162,A 39.3537,B 15.9089,C -0.281,E1 16.0332,E2 409.9629} C_DIS
LIN {X 102.7702,Y 83.2038,Z 162,A 37.4827,B 15.9089,C -0.2775,E1 16.0366,E2 411.8325} C_DIS
LIN {X 105.52,Y 79.6873,Z 162,A 35.5536,B 15.9089,C -0.2732,E1 16.0398,E2 413.7624} C_DIS
LIN {X 108.0137,Y 76.2731,Z 162,A 33.8221,B 15.909,C -0.2723,E1 16.0427,E2 415.4834} C_DIS
LIN {X 110.3121,Y 72.9098,Z 162,A 32.0624,B 15.909,C -0.2681,E1 16.0454,E2 417.2439} C_DIS
LIN {X 112.5427,Y 69.4175,Z 162,A 30.2315,B 15.9092,C -0.2624,E1 16.0481,E2 419.0805} C_DIS
LIN {X 114.3393,Y 66.4161,Z 162,A 28.7465,B 15.9092,C -0.2596,E1 16.0502,E2 420.5631} C_DIS
LIN {X 116.4284,Y 62.6816,Z 162,A 26.9238,B 15.9092,C -0.2558,E1 16.0527,E2 422.3838} C_DIS
LIN {X 118.2116,Y 59.251,Z 162,A 24.8084,B 15.9096,C -0.2359,E1 16.0554,E2 424.5529} C_DIS
LIN {X 120.0518,Y 55.4219,Z 162,A 23.5047,B 15.9094,C -0.2499,E1 16.0569,E2 425.7946} C_DIS
LIN {X 121.3808,Y 52.4474,Z 162,A 22.0721,B 15.9094,C -0.2453,E1 16.0585,E2 427.2312} C_DIS
LIN {X 122.7401,Y 49.1831,Z 162,A 20.5602,B 15.9094,C -0.2417,E1 16.0601,E2 428.7422} C_DIS
LIN {X 124.0543,Y 45.7712,Z 162,A 18.98,B 15.9095,C -0.2374,E1 16.0616,E2 430.3237} C_DIS
LIN {X 126.0794,Y 39.8522,Z 162,A 15.7276,B 15.9099,C -0.2105,E1 16.0645,E2 433.6432} C_DIS
LIN {X 127.4504,Y 35.2224,Z 162,A 14.428,B 15.9096,C -0.2326,E1 16.0655,E2 434.8508} C_DIS
LIN {X 128.8716,Y 29.601,Z 162,A 11.2477,B 15.91,C -0.2015,E1 16.0676,E2 438.1137} C_DIS
LIN {X 129.7936,Y 25.2568,Z 162,A 10.0182,B 15.9098,C -0.2205,E1 16.0683,E2 439.2627} C_DIS
LIN {X 130.4355,Y 21.6957,Z 162,A 8.3049,B 15.9099,C -0.2106,E1 16.0691,E2 440.9953} C_DIS
LIN {X 130.9906,Y 18.0559,Z 162,A 6.6108,B 15.91,C -0.2023,E1 16.0698,E2 442.7031} C_DIS
LIN {X 131.4776,Y 14.0633,Z 162,A 4.9942,B 15.91,C -0.2016,E1 16.0703,E2 444.3068} C_DIS
LIN {X 131.8392,Y 10.1409,Z 162,A 3.2583,B 15.9101,C -0.1954,E1 16.0707,E2 446.0483} C_DIS
LIN {X 132.0676,Y 6.5056,Z 162,A 1.7692,B 15.9101,C -0.1938,E1 16.0709,E2 447.5287} C_DIS
LIN {X 132.1913,Y 3.1455,Z 162,A 0.185,B 15.9102,C -0.1848,E1 16.0711,E2 449.1301} C_DIS
LIN {X 132.2265,Y -0.7398,Z 162,A -1.486,B 15.9102,C -0.1802,E1 16.0711,E2 450.8017} C_DIS
LIN {X 132.1256,Y -5.1945,Z 162,A -3.2748,B 15.9102,C -0.1794,E1 16.0709,E2 452.5761} C_DIS
LIN {X 131.9092,Y -9.1816,Z 162,A -5.0466,B 15.9104,C -0.1726,E1 16.0706,E2 454.3551} C_DIS
LIN {X 131.6038,Y -12.8299,Z 162,A -6.5601,B 15.9104,C -0.1704,E1 16.0702,E2 455.862} C_DIS
LIN {X 131.2014,Y -16.4575,Z 162,A -8.2515,B 15.9104,C -0.1616,E1 16.0697,E2 457.5688} C_DIS
LIN {X 130.6254,Y -20.5234,Z 162,A -9.9284,B 15.9104,C -0.1599,E1 16.069,E2 459.2358} C_DIS
LIN {X 129.9843,Y -24.2596,Z 162,A -11.4897,B 15.9105,C -0.1579,E1 16.0682,E2 460.7896} C_DIS
LIN {X 128.5387,Y -31.0143,Z 162,A -14.1404,B 15.9105,C -0.1612,E1 16.0667,E2 463.4031} C_DIS
LIN {X 127.1841,Y -36.1748,Z 162,A -16.7541,B 15.9106,C -0.1434,E1 16.0648,E2 466.0564} C_DIS
LIN {X 126.416,Y -38.7692,Z 162,A -17.9371,B 15.9106,C -0.1396,E1 16.0638,E2 467.2423} C_DIS
LIN {X 125.3875,Y -41.9771,Z 162,A -19.3793,B 15.9107,C -0.1359,E1 16.0626,E2 468.6845} C_DIS
LIN {X 124.1417,Y -45.5349,Z 162,A -21.0807,B 15.9107,C -0.1287,E1 16.0609,E2 470.3964} C_DIS
LIN {X 122.3042,Y -50.2619,Z 162,A -23.1293,B 15.9107,C -0.1277,E1 16.0589,E2 472.4301} C_DIS
LIN {X 121.2162,Y -52.8282,Z 162,A -24.3323,B 15.9107,C -0.1245,E1 16.0575,E2 473.6342} C_DIS
LIN {X 119.9652,Y -55.6093,Z 162,A -26.054,B 15.9109,C -0.1064,E1 16.0555,E2 475.4058} C_DIS
LIN {X 118.3422,Y -58.9867,Z 162,A -27.4112,B 15.9109,C -0.1114,E1 16.0538,E2 476.7333} C_DIS
LIN {X 115.622,Y -64.1569,Z 162,A -29.7636,B 15.9109,C -0.1108,E1 16.0507,E2 479.0676} C_DIS
LIN {X 113.7886,Y -67.3562,Z 162,A -31.4769,B 15.9109,C -0.1023,E1 16.0483,E2 480.7971} C_DIS
LIN {X 111.6,Y -70.9235,Z 162,A -33.9841,B 15.9111,C -0.073,E1 16.0444,E2 483.3899} C_DIS
LIN {X 108.3188,Y -75.8401,Z 162,A -35.5715,B 15.911,C -0.1008,E1 16.0421,E2 484.864} C_DIS
LIN {X 106.452,Y -78.4381,Z 162,A -37.7774,B 15.9111,C -0.0682,E1 16.0383,E2 487.1702} C_DIS
LIN {X 103.223,Y -82.642,Z 162,A -39.1947,B 15.9111,C -0.0936,E1 16.036,E2 488.4848} C_DIS
LIN {X 98.6763,Y -88.0204,Z 162,A -42.4377,B 15.9111,C -0.0794,E1 16.0301,E2 491.7552} C_DIS
LIN {X 95.7755,Y -91.1683,Z 162,A -44.347,B 15.9111,C -0.0732,E1 16.0264,E2 493.6734} C_DIS
LIN {X 92.9889,Y -94.0087,Z 162,A -46.6308,B 15.9111,C -0.0497,E1 16.0218,E2 496.0266} C_DIS
LIN {X 89.1665,Y -97.6425,Z 162,A -48.0873,B 15.9111,C -0.0737,E1 16.019,E2 497.3863} C_DIS
LIN {X 86.7143,Y -99.8262,Z 162,A -50.0891,B 15.9111,C -0.0504,E1 16.0146,E2 499.4596} C_DIS
LIN {X 83.606,Y -102.4431,Z 162,A -51.1967,B 15.9111,C -0.0696,E1 16.0124,E2 500.4907} C_DIS
LIN {X 81.2366,Y -104.3322,Z 162,A -52.7112,B 15.9111,C -0.0599,E1 16.009,E2 502.0311} C_DIS
LIN {X 79.1541,Y -105.9208,Z 162,A -53.9276,B 15.9111,C -0.0548,E1 16.0063,E2 503.2587} C_DIS
LIN {X 71.4279,Y -111.2772,Z 162,A -57.9544,B 15.9112,C -0.0489,E1 15.997,E2 507.2845} C_DIS
LIN {X 67.6579,Y -113.6088,Z 162,A -59.8445,B 15.9112,C -0.0467,E1 15.9925,E2 509.173} C_DIS
LIN {X 61.4895,Y -117.06,Z 162,A -62.7264,B 15.9112,C -0.048,E1 15.9855,E2 512.0363} C_DIS
LIN {X 55.1697,Y -120.1684,Z 162,A -65.8686,B 15.9112,C -0.0404,E1 15.9776,E2 515.1926} C_DIS
LIN {X 52.1946,Y -121.4901,Z 162,A -67.2825,B 15.9112,C -0.0383,E1 15.9739,E2 516.6083} C_DIS
LIN {X 49.1596,Y -122.7496,Z 162,A -68.6612,B 15.9112,C -0.038,E1 15.9704,E2 517.9829} C_DIS
LIN {X 45.9765,Y -123.9774,Z 162,A -70.1234,B 15.9112,C -0.0368,E1 15.9666,E2 519.4446} C_DIS
LIN {X 42.7414,Y -125.1303,Z 162,A -71.8283,B 15.9112,C -0.0277,E1 15.962,E2 521.1769} C_DIS
LIN {X 37.3624,Y -126.8391,Z 162,A -73.9512,B 15.9112,C -0.0361,E1 15.9564,E2 523.2629} C_DIS
LIN {X 34.048,Y -127.7686,Z 162,A -75.601,B 15.9112,C -0.0293,E1 15.9519,E2 524.933} C_DIS
LIN {X 31.3019,Y -128.4694,Z 162,A -76.8613,B 15.9112,C -0.0271,E1 15.9485,E2 526.1982} C_DIS
LIN {X 26.9423,Y -129.4548,Z 162,A -78.767,B 15.9112,C -0.0266,E1 15.9433,E2 528.1018} C_DIS
LIN {X 23.3972,Y -130.141,Z 162,A -80.3312,B 15.9112,C -0.0255,E1 15.939,E2 529.667} C_DIS
LIN {X 19.0323,Y -130.8511,Z 162,A -82.2217,B 15.9112,C -0.0251,E1 15.9338,E2 531.5557} C_DIS
LIN {X 15.4925,Y -131.3169,Z 162,A -83.7244,B 15.9112,C -0.0258,E1 15.9296,E2 533.054} C_DIS
LIN {X 11.5508,Y -131.7228,Z 162,A -85.4849,B 15.9112,C -0.0235,E1 15.9247,E2 534.8208} C_DIS
LIN {X 7.8219,Y -131.9965,Z 162,A -87.1497,B 15.9112,C -0.0215,E1 15.9201,E2 536.492} C_DIS
LIN {X 3.6135,Y -132.1783,Z 162,A -88.8562,B 15.9112,C -0.0249,E1 15.9154,E2 538.1851} C_DIS
LIN {X 0.913,Y -132.2218,Z 162,A -89.6324,B 15.9112,C -0.0378,E1 15.9133,E2 538.9141} C_DIS
Enddeposition()
LIN {X 0.913,Y -132.2218,Z 162,A -89.6324,B 15.9112,C -0.0378,E1 15.9133,E2 538.9141} C_DIS
Startdeposition()
$VEL.CP = VEL_PRINT
LIN {X 2.6378,Y -131.2793,Z 162,A -87.7972,B 13.3999,C 0.1357,E1 13.4059,E2 537.6924} C_DIS
LIN {X 6.6265,Y -131.1376,Z 162,A -86.121,B 13.3999,C 0.137,E1 13.4106,E2 536.0232} C_DIS
LIN {X 10.7097,Y -130.8678,Z 162,A -84.2688,B 13.3999,C 0.1345,E1 13.4158,E2 534.1619} C_DIS
LIN {X 14.7773,Y -130.4727,Z 162,A -82.4775,B 13.3999,C 0.1335,E1 13.4207,E2 532.3687} C_DIS
LIN {X 18.5154,Y -129.9928,Z 162,A -80.9302,B 13.3999,C 0.1353,E1 13.425,E2 530.832} C_DIS
LIN {X 22.2124,Y -129.4137,Z 162,A -79.1774,B 13.3999,C 0.1309,E1 13.4299,E2 529.0637} C_DIS
LIN {X 26.3528,Y -128.6331,Z 162,A -77.5237,B 13.3999,C 0.1349,E1 13.4343,E2 527.431} C_DIS
LIN {X 29.8966,Y -127.8576,Z 162,A -75.9007,B 13.3999,C 0.1325,E1 13.4388,E2 525.8021} C_DIS
LIN {X 33.1322,Y -127.0578,Z 162,A -74.3507,B 13.4,C 0.1284,E1 13.443,E2 524.2394} C_DIS
LIN {X 37.8466,Y -125.7334,Z 162,A -71.8746,B 13.4001,C 0.1164,E1 13.4497,E2 521.7203} C_DIS
LIN {X 41.5601,Y -124.5538,Z 162,A -70.6475,B 13.4001,C 0.1284,E1 13.4529,E2 520.5493} C_DIS
LIN {X 44.4865,Y -123.5387,Z 162,A -69.2507,B 13.4001,C 0.1256,E1 13.4565,E2 519.146} C_DIS
LIN {X 48.032,Y -122.2049,Z 162,A -67.6273,B 13.4001,C 0.1245,E1 13.4608,E2 517.5248} C_DIS
LIN {X 51.8587,Y -120.63,Z 162,A -65.7965,B 13.4001,C 0.1214,E1 13.4655,E2 515.6893} C_DIS
LIN {X 54.8489,Y -119.3002,Z 162,A -64.2517,B 13.4001,C 0.116,E1 13.4695,E2 514.129} C_DIS
LIN {X 59.1961,Y -117.2042,Z 162,A -62.2606,B 13.4001,C 0.1163,E1 13.4744,E2 512.1498} C_DIS
LIN {X 62.3689,Y -115.5489,Z 162,A -60.9362,B 13.4001,C 0.121,E1 13.4776,E2 510.8527} C_DIS
LIN {X 65.507,Y -113.7994,Z 162,A -59.132,B 13.4001,C 0.1115,E1 13.4821,E2 509.0183} C_DIS
LIN {X 69.0479,Y -111.6866,Z 162,A -57.2879,B 13.4001,C 0.1072,E1 13.4865,E2 507.1669} C_DIS
LIN {X 72.2972,Y -109.6107,Z 162,A -55.4014,B 13.4003,C 0.0981,E1 13.491,E2 505.2539} C_DIS
LIN {X 75.2207,Y -107.6256,Z 162,A -54.2148,B 13.4002,C 0.1059,E1 13.4936,E2 504.1089} C_DIS
LIN {X 78.2335,Y -105.4559,Z 162,A -52.52,B 13.4002,C 0.1007,E1 13.4974,E2 502.4033} C_DIS
LIN {X 81.7026,Y -102.7913,Z 162,A -50.8247,B 13.4002,C 0.1034,E1 13.5011,E2 500.7318} C_DIS
LIN {X 84.3204,Y -100.655,Z 162,A -48.6399,B 13.4004,C 0.0789,E1 13.506,E2 498.4589} C_DIS
LIN {X 88.018,Y -97.4385,Z 162,A -47.2394,B 13.4003,C 0.0968,E1 13.5087,E2 497.1459} C_DIS
LIN {X 93.0599,Y -92.6349,Z 162,A -43.775,B 13.4003,C 0.0773,E1 13.5158,E2 493.6263} C_DIS
LIN {X 95.4822,Y -90.136,Z 162,A -42.6466,B 13.4003,C 0.0858,E1 13.5179,E2 492.5436} C_DIS
LIN {X 98.0837,Y -87.2989,Z 162,A -41.0206,B 13.4003,C 0.0835,E1 13.5209,E2 490.9221} C_DIS
LIN {X 101.4384,Y -83.377,Z 162,A -38.5064,B 13.4004,C 0.0702,E1 13.5255,E2 488.3735} C_DIS
LIN {X 105.1165,Y -78.6892,Z 162,A -36.0528,B 13.4004,C 0.0683,E1 13.5296,E2 485.9346} C_DIS
LIN {X 107.5827,Y -75.2824,Z 162,A -34.2475,B 13.4004,C 0.0647,E1 13.5326,E2 484.1307} C_DIS
LIN {X 110.8707,Y -70.3501,Z 162,A -31.6485,B 13.4004,C 0.0576,E1 13.5365,E2 481.5269} C_DIS
LIN {X 113.2369,Y -66.4739,Z 162,A -29.7916,B 13.4004,C 0.0563,E1 13.5392,E2 479.6828} C_DIS
LIN {X 115.1435,Y -63.1143,Z 162,A -28.0279,B 13.4005,C 0.0493,E1 13.5416,E2 477.9075} C_DIS
LIN {X 116.7856,Y -60.0184,Z 162,A -26.6247,B 13.4005,C 0.0491,E1 13.5434,E2 476.5176} C_DIS
LIN {X 118.7455,Y -56.0423,Z 162,A -24.5675,B 13.4005,C 0.04,E1 13.5459,E2 474.4432} C_DIS
LIN {X 120.4095,Y -52.3688,Z 162,A -22.9445,B 13.4005,C 0.0393,E1 13.5477,E2 472.8345} C_DIS
LIN {X 122.7892,Y -46.5179,Z 162,A -20.1844,B 13.4005,C 0.0314,E1 13.5506,E2 470.0705} C_DIS
LIN {X 123.9883,Y -43.2183,Z 162,A -18.7468,B 13.4005,C 0.03,E1 13.5519,E2 468.6424} C_DIS
LIN {X 124.9782,Y -40.267,Z 162,A -17.3676,B 13.4005,C 0.0254,E1 13.5531,E2 467.259} C_DIS
LIN {X 125.9156,Y -37.2327,Z 162,A -16.1318,B 13.4005,C 0.026,E1 13.5541,E2 466.0395} C_DIS
LIN {X 127.2961,Y -32.1965,Z 162,A -13.7312,B 13.4005,C 0.0156,E1 13.5559,E2 463.6214} C_DIS
LIN {X 128.8468,Y -25.2953,Z 162,A -10.7159,B 13.4006,C 0.0088,E1 13.5576,E2 460.6112} C_DIS
LIN {X 129.6609,Y -20.722,Z 162,A -8.5846,B 13.4006,C -0.0004,E1 13.5586,E2 458.4648} C_DIS
LIN {X 130.1997,Y -16.9998,Z 162,A -7.0473,B 13.4006,C -0.0021,E1 13.5592,E2 456.9379} C_DIS
LIN {X 130.672,Y -12.8802,Z 162,A -5.2171,B 13.4006,C -0.0082,E1 13.5598,E2 455.1032} C_DIS
LIN {X 131.0152,Y -8.7434,Z 162,A -3.3862,B 13.4006,C -0.0142,E1 13.5601,E2 453.2678} C_DIS
LIN {X 131.2305,Y -4.4686,Z 162,A -1.5626,B 13.4006,C -0.0184,E1 13.5604,E2 451.4473} C_DIS
LIN {X 131.3033,Y -0.8067,Z 162,A -0.1069,B 13.4006,C -0.0187,E1 13.5604,E2 450.0068} C_DIS
LIN {X 131.2771,Y 2.7673,Z 162,A 1.5499,B 13.4006,C -0.0264,E1 13.5604,E2 448.3366} C_DIS
LIN {X 131.1324,Y 6.729,Z 162,A 3.2528,B 13.4006,C -0.0307,E1 13.5601,E2 446.6349} C_DIS
LIN {X 130.8458,Y 10.9704,Z 162,A 5.0286,B 13.4006,C -0.0338,E1 13.5598,E2 444.8665} C_DIS
LIN {X 130.4726,Y 14.7786,Z 162,A 6.8107,B 13.4006,C -0.0422,E1 13.5592,E2 443.0692} C_DIS
LIN {X 129.9429,Y 18.8648,Z 162,A 8.5514,B 13.4006,C -0.0457,E1 13.5586,E2 441.3334} C_DIS
LIN {X 129.2761,Y 22.9924,Z 162,A 10.2342,B 13.4006,C -0.0467,E1 13.5578,E2 439.6657} C_DIS
LIN {X 127.9331,Y 29.5657,Z 162,A 13.1764,B 13.4005,C -0.0556,E1 13.5561,E2 436.7188} C_DIS
LIN {X 126.9669,Y 33.473,Z 162,A 14.9211,B 13.4005,C -0.0603,E1 13.5549,E2 434.9737} C_DIS
LIN {X 126.0716,Y 36.6998,Z 162,A 16.3767,B 13.4005,C -0.0643,E1 13.5538,E2 433.5174} C_DIS
LIN {X 123.7611,Y 43.8698,Z 162,A 19.6921,B 13.4005,C -0.0743,E1 13.5508,E2 430.1957} C_DIS
LIN {X 122.5853,Y 47.0535,Z 162,A 21.1053,B 13.4004,C -0.0763,E1 13.5494,E2 428.7892} C_DIS
LIN {X 121.3162,Y 50.2334,Z 162,A 22.5246,B 13.4004,C -0.0781,E1 13.548,E2 427.3775} C_DIS
LIN {X 119.9329,Y 53.4506,Z 162,A 24.0217,B 13.4004,C -0.0813,E1 13.5463,E2 425.8827} C_DIS
LIN {X 118.0737,Y 57.4452,Z 162,A 26.0843,B 13.4004,C -0.0906,E1 13.5438,E2 423.8019} C_DIS
LIN {X 116.1998,Y 61.1428,Z 162,A 27.6856,B 13.4004,C -0.0891,E1 13.5418,E2 422.2238} C_DIS
LIN {X 114.4191,Y 64.4178,Z 162,A 29.443,B 13.4003,C -0.0972,E1 13.5394,E2 420.4496} C_DIS
LIN {X 112.3002,Y 68.0444,Z 162,A 31.2338,B 13.4003,C -0.1005,E1 13.5368,E2 418.6625} C_DIS
LIN {X 109.9361,Y 71.8021,Z 162,A 33.1912,B 13.4002,C -0.1059,E1 13.5339,E2 416.7013} C_DIS
LIN {X 107.1555,Y 75.8888,Z 162,A 35.6053,B 13.4001,C -0.1188,E1 13.5299,E2 414.2551} C_DIS
LIN {X 104.9633,Y 78.8931,Z 162,A 36.9426,B 13.4001,C -0.114,E1 13.5278,E2 412.9508} C_DIS
LIN {X 102.2116,Y 82.4266,Z 162,A 38.8339,B 13.4001,C -0.1166,E1 13.5245,E2 411.0658} C_DIS
LIN {X 99.318,Y 85.8916,Z 162,A 40.806,B 13.4001,C -0.121,E1 13.5209,E2 409.0923} C_DIS
LIN {X 96.3616,Y 89.1962,Z 162,A 42.7612,B 13.4001,C -0.1258,E1 13.5172,E2 407.1337} C_DIS
LIN {X 93.2214,Y 92.4724,Z 162,A 44.6649,B 13.4001,C -0.1276,E1 13.5135,E2 405.2381} C_DIS
LIN {X 90.2751,Y 95.351,Z 162,A 46.4924,B 13.4,C -0.1321,E1 13.5099,E2 403.4063} C_DIS
LIN {X 86.9381,Y 98.4028,Z 162,A 48.4148,B 13.4,C -0.1344,E1 13.5059,E2 401.489} C_DIS
LIN {X 83.5121,Y 101.3271,Z 162,A 50.3912,B 13.4,C -0.1384,E1 13.5016,E2 399.5106} C_DIS
LIN {X 80.1086,Y 104.0392,Z 162,A 52.3035,B 13.3999,C -0.1421,E1 13.4974,E2 397.596} C_DIS
LIN {X 76.5893,Y 106.656,Z 162,A 53.9804,B 13.3999,C -0.1385,E1 13.4937,E2 395.9466} C_DIS
LIN {X 73.6971,Y 108.6744,Z 162,A 56.0295,B 13.3997,C -0.1558,E1 13.4889,E2 393.8366} C_DIS
LIN {X 70.4274,Y 110.822,Z 162,A 57.4389,B 13.3997,C -0.1498,E1 13.4856,E2 392.4622} C_DIS
LIN {X 66.6896,Y 113.1101,Z 162,A 59.3384,B 13.3997,C -0.1522,E1 13.4811,E2 390.5638} C_DIS
LIN {X 63.0928,Y 115.1552,Z 162,A 61.0409,B 13.3997,C -0.1517,E1 13.4769,E2 388.8733} C_DIS
LIN {X 59.8461,Y 116.8733,Z 162,A 62.4242,B 13.3998,C -0.1476,E1 13.4736,E2 387.5156} C_DIS
LIN {X 57.2531,Y 118.167,Z 162,A 63.9475,B 13.3998,C -0.1565,E1 13.4697,E2 385.9617} C_DIS
LIN {X 53.9309,Y 119.7181,Z 162,A 65.4375,B 13.3998,C -0.1553,E1 13.4659,E2 384.4846} C_DIS
LIN {X 50.8434,Y 121.0615,Z 162,A 66.914,B 13.3998,C -0.1571,E1 13.4621,E2 383.0072} C_DIS
LIN {X 47.9095,Y 122.2525,Z 162,A 68.2994,B 13.3997,C -0.1586,E1 13.4585,E2 381.6213} C_DIS
LIN {X 44.4886,Y 123.538,Z 162,A 69.8736,B 13.3997,C -0.1596,E1 13.4544,E2 380.0497} C_DIS
LIN {X 41.1265,Y 124.6982,Z 162,A 71.5133,B 13.3997,C -0.1634,E1 13.4501,E2 378.3998} C_DIS
LIN {X 37.1026,Y 125.9537,Z 162,A 73.011,B 13.3997,C -0.1553,E1 13.4462,E2 376.9423} C_DIS
LIN {X 33.2213,Y 127.034,Z 162,A 75.0478,B 13.3997,C -0.1643,E1 13.4406,E2 374.8732} C_DIS
LIN {X 29.5956,Y 127.9263,Z 162,A 76.63,B 13.3997,C -0.164,E1 13.4363,E2 373.2969} C_DIS
LIN {X 26.8542,Y 128.5311,Z 162,A 78.3802,B 13.3994,C -0.1793,E1 13.4314,E2 371.4851} C_DIS
LIN {X 22.5921,Y 129.3477,Z 162,A 79.8687,B 13.3996,C -0.1688,E1 13.4274,E2 370.0449} C_DIS
LIN {X 18.7279,Y 129.9624,Z 162,A 81.4284,B 13.3996,C -0.1654,E1 13.4231,E2 368.503} C_DIS
LIN {X 15.2708,Y 130.4141,Z 162,A 83.038,B 13.3996,C -0.1683,E1 13.4187,E2 366.8835} C_DIS
LIN {X 11.1309,Y 130.8322,Z 162,A 84.801,B 13.3996,C -0.1672,E1 13.4138,E2 365.1274} C_DIS
LIN {X 7.1408,Y 131.1117,Z 162,A 86.5889,B 13.3996,C -0.1685,E1 13.4088,E2 363.3352} C_DIS
LIN {X 3.6977,Y 131.2529,Z 162,A 88.095,B 13.3996,C -0.1686,E1 13.4046,E2 361.8294} C_DIS
LIN {X -0.2727,Y 131.3055,Z 162,A 89.8699,B 13.3996,C -0.1697,E1 13.3996,E2 360.0504} C_DIS
LIN {X -4.6318,Y 131.2241,Z 162,A 91.7416,B 13.3996,C -0.1685,E1 13.3944,E2 358.1833} C_DIS
LIN {X -8.3235,Y 131.0411,Z 162,A 93.3732,B 13.3996,C -0.1687,E1 13.3898,E2 356.5503} C_DIS
LIN {X -12.4668,Y 130.7117,Z 162,A 95.1067,B 13.3996,C -0.1659,E1 13.385,E2 354.8273} C_DIS
LIN {X -16.138,Y 130.3106,Z 162,A 96.7877,B 13.3996,C -0.1671,E1 13.3804,E2 353.1392} C_DIS
LIN {X -20.0068,Y 129.7716,Z 162,A 98.2931,B 13.3996,C -0.1609,E1 13.3763,E2 351.658} C_DIS
LIN {X -26.6813,Y 128.5663,Z 162,A 101.3473,B 13.3996,C -0.1615,E1 13.3679,E2 348.595} C_DIS
LIN {X -33.1984,Y 127.0401,Z 162,A 104.3994,B 13.3996,C -0.1627,E1 13.3596,E2 345.5297} C_DIS
LIN {X -36.5943,Y 126.1025,Z 162,A 105.8741,B 13.3996,C -0.1597,E1 13.3556,E2 344.0635} C_DIS
LIN {X -39.4258,Y 125.2469,Z 162,A 107.8696,B 13.3995,C -0.177,E1 13.3501,E2 341.9863} C_DIS
LIN {X -44.4093,Y 123.5666,Z 162,A 109.504,B 13.3997,C -0.1572,E1 13.346,E2 340.4314} C_DIS
LIN {X -47.6953,Y 122.3358,Z 162,A 111.0564,B 13.3997,C -0.156,E1 13.3419,E2 338.8779} C_DIS
LIN {X -51.8408,Y 120.6377,Z 162,A 113.3159,B 13.3997,C -0.1615,E1 13.336,E2 336.5844} C_DIS
LIN {X -54.9967,Y 119.2318,Z 162,A 114.4645,B 13.3997,C -0.1503,E1 13.3332,E2 335.4792} C_DIS
LIN {X -58.0616,Y 117.7696,Z 162,A 115.9117,B 13.3998,C -0.1473,E1 13.3296,E2 334.0373} C_DIS
LIN {X -64.6699,Y 114.2773,Z 162,A 119.3713,B 13.3998,C -0.1475,E1 13.3211,E2 330.558} C_DIS
LIN {X -68.294,Y 112.1492,Z 162,A 121.2083,B 13.3998,C -0.1447,E1 13.3166,E2 328.7225} C_DIS
LIN {X -70.7257,Y 110.6311,Z 162,A 122.5671,B 13.3998,C -0.1453,E1 13.3134,E2 327.3522} C_DIS
LIN {X -74.634,Y 108.0338,Z 162,A 124.9871,B 13.3998,C -0.1512,E1 13.3078,E2 324.8907} C_DIS
LIN {X -78.3374,Y 105.3785,Z 162,A 126.5114,B 13.3999,C -0.1358,E1 13.3045,E2 323.423} C_DIS
LIN {X -81.9355,Y 102.6059,Z 162,A 128.464,B 13.3999,C -0.1313,E1 13.3002,E2 321.476} C_DIS
LIN {X -85.9135,Y 99.2992,Z 162,A 130.7855,B 13.4,C -0.1284,E1 13.2952,E2 319.1495} C_DIS
LIN {X -89.1167,Y 96.4349,Z 162,A 132.6665,B 13.4,C -0.1247,E1 13.2913,E2 317.2699} C_DIS
LIN {X -92.161,Y 93.5297,Z 162,A 134.3928,B 13.4,C -0.118,E1 13.2879,E2 315.5585} C_DIS
LIN {X -94.3939,Y 91.2752,Z 162,A 135.9292,B 13.4,C -0.1188,E1 13.2849,E2 314.0059} C_DIS
LIN {X -97.4075,Y 88.0522,Z 162,A 137.8579,B 13.4001,C -0.1145,E1 13.2812,E2 312.0791} C_DIS
LIN {X -100.1911,Y 84.8714,Z 162,A 139.7317,B 13.4001,C -0.111,E1 13.2778,E2 310.2041} C_DIS
LIN {X -103.1171,Y 81.2913,Z 162,A 141.7743,B 13.4001,C -0.1068,E1 13.2742,E2 308.161} C_DIS
LIN {X -105.7772,Y 77.7981,Z 162,A 143.6591,B 13.4002,C -0.1013,E1 13.2711,E2 306.2821} C_DIS
LIN {X -108.0294,Y 74.6404,Z 162,A 145.2758,B 13.4002,C -0.0953,E1 13.2685,E2 304.6763} C_DIS
LIN {X -110.0403,Y 71.6416,Z 162,A 147.0127,B 13.4002,C -0.0953,E1 13.2658,E2 302.9225} C_DIS
LIN {X -112.4923,Y 67.7267,Z 162,A 149.1144,B 13.4002,C -0.0921,E1 13.2627,E2 300.8132} C_DIS
LIN {X -114.9196,Y 63.5206,Z 162,A 151.0779,B 13.4004,C -0.0827,E1 13.2601,E2 298.8704} C_DIS
LIN {X -117.0638,Y 59.472,Z 162,A 153.1616,B 13.4004,C -0.0794,E1 13.2574,E2 296.7792} C_DIS
LIN {X -119.0093,Y 55.478,Z 162,A 155.0491,B 13.4004,C -0.0729,E1 13.2551,E2 294.9002} C_DIS
LIN {X -120.4274,Y 52.3274,Z 162,A 156.5688,B 13.4004,C -0.069,E1 13.2534,E2 293.3809} C_DIS
LIN {X -121.7338,Y 49.2114,Z 162,A 158.073,B 13.4004,C -0.0656,E1 13.2518,E2 291.875} C_DIS
LIN {X -123.5001,Y 44.5937,Z 162,A 160.2706,B 13.4004,C -0.0605,E1 13.2496,E2 289.6754} C_DIS
LIN {X -124.6065,Y 41.4016,Z 162,A 161.729,B 13.4004,C -0.0559,E1 13.2483,E2 288.2207} C_DIS
LIN {X -125.7723,Y 37.7196,Z 162,A 163.4309,B 13.4005,C -0.0515,E1 13.2469,E2 286.519} C_DIS
LIN {X -126.7295,Y 34.3631,Z 162,A 165.0762,B 13.4005,C -0.05,E1 13.2457,E2 284.8612} C_DIS
LIN {X -127.6655,Y 30.6992,Z 162,A 166.6701,B 13.4005,C -0.0438,E1 13.2446,E2 283.2759} C_DIS
LIN {X -128.6663,Y 26.1899,Z 162,A 168.7125,B 13.4005,C -0.0386,E1 13.2434,E2 281.2328} C_DIS
LIN {X -129.2179,Y 23.3174,Z 162,A 170.2047,B 13.4005,C -0.04,E1 13.2427,E2 279.7168} C_DIS
LIN {X -130.0023,Y 18.4488,Z 162,A 172.1716,B 13.4005,C -0.0292,E1 13.2419,E2 277.7742} C_DIS
LIN {X -130.4833,Y 14.6784,Z 162,A 173.9501,B 13.4005,C -0.0271,E1 13.2413,E2 275.9838} C_DIS
LIN {X -130.8684,Y 10.7024,Z 162,A 175.7259,B 13.4005,C -0.0228,E1 13.2408,E2 274.2061} C_DIS
LIN {X -131.1818,Y 5.7172,Z 162,A 178.6359,B 13.4005,C -0.0341,E1 13.2405,E2 271.2121} C_DIS
LIN {X -131.3073,Y -0.1892,Z 162,A -178.7885,B 13.4005,C -0.0264,E1 13.2405,E2 268.6397} C_DIS
LIN {X -131.176,Y -5.8624,Z 162,A -177.0098,B 13.4006,C -0.0019,E1 13.2406,E2 266.9467} C_DIS
LIN {X -130.7313,Y -12.2616,Z 162,A -174.1381,B 13.4006,C 0.0046,E1 13.2413,E2 264.0695} C_DIS
LIN {X -129.8886,Y -19.2442,Z 162,A -171.0169,B 13.4006,C 0.0124,E1 13.2424,E2 260.9456} C_DIS
LIN {X -129.2422,Y -23.1816,Z 162,A -169.3232,B 13.4006,C 0.0186,E1 13.2432,E2 259.2593} C_DIS
LIN {X -128.2685,Y -28.0755,Z 162,A -167.0562,B 13.4006,C 0.0227,E1 13.2445,E2 256.9839} C_DIS
LIN {X -127.3221,Y -32.0943,Z 162,A -165.3201,B 13.4006,C 0.0295,E1 13.2456,E2 255.2574} C_DIS
LIN {X -126.4785,Y -35.2716,Z 162,A -163.8795,B 13.4006,C 0.0334,E1 13.2467,E2 253.8175} C_DIS
LIN {X -125.3492,Y -39.1021,Z 162,A -162.0196,B 13.4006,C 0.0355,E1 13.2482,E2 251.9455} C_DIS
LIN {X -124.1156,Y -42.8511,Z 162,A -160.4504,B 13.4006,C 0.044,E1 13.2496,E2 250.3959} C_DIS
LIN {X -123.0754,Y -45.7538,Z 162,A -159.1099,B 13.4006,C 0.0479,E1 13.2509,E2 249.0573} C_DIS
LIN {X -122.2756,Y -47.85,Z 162,A -157.7872,B 13.4006,C 0.0421,E1 13.2522,E2 247.6947} C_DIS
LIN {X -120.2325,Y -52.7781,Z 162,A -154.6732,B 13.4006,C 0.0287,E1 13.2559,E2 244.4885} C_DIS
LIN {X -117.3071,Y -58.9941,Z 162,A -152.6217,B 13.4005,C 0.0603,E1 13.2582,E2 242.553} C_DIS
LIN {X -115.4707,Y -62.5144,Z 162,A -150.7805,B 13.4005,C 0.062,E1 13.2606,E2 240.7003} C_DIS
LIN {X -113.2399,Y -66.4688,Z 162,A -148.814,B 13.4005,C 0.0674,E1 13.2634,E2 238.737} C_DIS
LIN {X -110.9928,Y -70.1567,Z 162,A -147.0055,B 13.4005,C 0.0739,E1 13.266,E2 236.9389} C_DIS
LIN {X -108.8088,Y -73.4984,Z 162,A -145.1873,B 13.4004,C 0.0762,E1 13.2689,E2 235.1129} C_DIS
LIN {X -106.398,Y -76.9471,Z 162,A -143.3022,B 13.4004,C 0.0793,E1 13.2719,E2 233.2232} C_DIS
LIN {X -103.7833,Y -80.4387,Z 162,A -141.4324,B 13.4004,C 0.0845,E1 13.2751,E2 231.3585} C_DIS
LIN {X -100.8015,Y -84.1459,Z 162,A -139.4633,B 13.4003,C 0.0919,E1 13.2785,E2 229.4034} C_DIS
LIN {X -95.9194,Y -89.671,Z 162,A -136.0569,B 13.4003,C 0.0939,E1 13.2849,E2 225.9763} C_DIS
LIN {X -92.8581,Y -92.838,Z 162,A -134.0704,B 13.4003,C 0.0962,E1 13.2888,E2 223.9831} C_DIS
LIN {X -90.0813,Y -95.5339,Z 162,A -132.1666,B 13.4003,C 0.094,E1 13.2927,E2 222.0542} C_DIS
LIN {X -87.5653,Y -97.8452,Z 162,A -129.6094,B 13.4004,C 0.0689,E1 13.2984,E2 219.3682} C_DIS
LIN {X -80.8034,Y -103.5003,Z 162,A -127.0218,B 13.4002,C 0.1087,E1 13.3037,E2 216.9348} C_DIS
LIN {X -78.1462,Y -105.5208,Z 162,A -125.555,B 13.4002,C 0.1109,E1 13.3069,E2 215.4672} C_DIS
LIN {X -74.7127,Y -107.9791,Z 162,A -123.6684,B 13.4002,C 0.1127,E1 13.3113,E2 213.5759} C_DIS
LIN {X -71.0802,Y -110.4042,Z 162,A -121.9326,B 13.4001,C 0.12,E1 13.3153,E2 211.8609} C_DIS
LIN {X -68.0738,Y -112.2824,Z 162,A -120.2773,B 13.4001,C 0.1194,E1 13.3192,E2 210.1928} C_DIS
LIN {X -64.7869,Y -114.2109,Z 162,A -118.597,B 13.4001,C 0.1212,E1 13.3233,E2 208.5108} C_DIS
LIN {X -61.4494,Y -116.0388,Z 162,A -117.1479,B 13.4,C 0.1289,E1 13.3268,E2 207.0871} C_DIS
LIN {X -58.44,Y -117.583,Z 162,A -115.4955,B 13.4,C 0.1261,E1 13.331,E2 205.4137} C_DIS
LIN {X -55.3779,Y -119.0555,Z 162,A -114.0127,B 13.4,C 0.1278,E1 13.3347,E2 203.931} C_DIS
LIN {X -52.2396,Y -120.4653,Z 162,A -112.4782,B 13.4,C 0.1285,E1 13.3387,E2 202.3925} C_DIS
LIN {X -49.2805,Y -121.7059,Z 162,A -111.0696,B 13.4,C 0.1297,E1 13.3423,E2 200.9829} C_DIS
LIN {X -46.0877,Y -122.9504,Z 162,A -109.6035,B 13.4,C 0.1318,E1 13.3461,E2 199.5202} C_DIS
LIN {X -42.8949,Y -124.1004,Z 162,A -108.1033,B 13.4,C 0.1326,E1 13.3501,E2 198.0176} C_DIS
LIN {X -39.2638,Y -125.2987,Z 162,A -106.1626,B 13.4,C 0.1265,E1 13.3553,E2 196.044} C_DIS
LIN {X -34.2612,Y -126.7567,Z 162,A -104.1459,B 13.4,C 0.135,E1 13.3607,E2 194.0579} C_DIS
LIN {X -30.3296,Y -127.7546,Z 162,A -101.9879,B 13.4,C 0.1254,E1 13.3666,E2 191.8527} C_DIS
LIN {X -26.6295,Y -128.5768,Z 162,A -100.657,B 13.4,C 0.1351,E1 13.3702,E2 190.5605} C_DIS
LIN {X -22.7633,Y -129.3171,Z 162,A -98.8944,B 13.4,C 0.1345,E1 13.375,E2 188.792} C_DIS
LIN {X -18.8584,Y -129.9438,Z 162,A -97.2407,B 13.4,C 0.137,E1 13.3796,E2 187.1465} C_DIS
LIN {X -15.184,Y -130.4244,Z 162,A -95.569,B 13.4,C 0.1359,E1 13.3842,E2 185.4676} C_DIS
LIN {X -11.5895,Y -130.7935,Z 162,A -93.9754,B 13.4,C 0.1356,E1 13.3887,E2 183.8715} C_DIS
LIN {X -7.2671,Y -131.1054,Z 162,A -92.0757,B 13.4,C 0.1355,E1 13.394,E2 181.9699} C_DIS
LIN {X -3.5333,Y -131.2575,Z 162,A -90.5429,B 13.4,C 0.1381,E1 13.3982,E2 180.4482} C_DIS
LIN {X 0.9021,Y -131.2997,Z 162,A -88.7167,B 13.3999,C 0.1409,E1 13.4033,E2 178.6342} C_DIS
Enddeposition()
LIN {X 0.9021,Y -131.2997,Z 162,A -88.7167,B 13.3999,C 0.1409,E1 13.4033,E2 178.6342} C_DIS
Startdeposition()
$VEL.CP = VEL_PRINT
LIN {X -0.6843,Y -130.3804,Z 162,A -90.0421,B 13.3995,C 0.1502,E1 13.3992,E2 179.9996} C_DIS
LIN {X -4.7994,Y -130.2941,Z 162,A -91.8237,B 13.3995,C 0.1496,E1 13.3942,E2 181.7787} C_DIS
LIN {X -8.6866,Y -130.0942,Z 162,A -93.6009,B 13.3995,C 0.1514,E1 13.3892,E2 183.5646} C_DIS
LIN {X -11.8714,Y -129.8419,Z 162,A -95.0091,B 13.3995,C 0.1514,E1 13.3853,E2 184.9738} C_DIS
LIN {X -15.2884,Y -129.4827,Z 162,A -96.4041,B 13.3995,C 0.1479,E1 13.3815,E2 186.3558} C_DIS
LIN {X -18.2179,Y -129.1032,Z 162,A -97.7945,B 13.3995,C 0.1501,E1 13.3776,E2 187.7576} C_DIS
LIN {X -21.6162,Y -128.5777,Z 162,A -99.2523,B 13.3995,C 0.1481,E1 13.3736,E2 189.2094} C_DIS
LIN {X -24.7749,Y -128.0068,Z 162,A -100.6703,B 13.3995,C 0.1478,E1 13.3697,E2 190.6287} C_DIS
LIN {X -27.9515,Y -127.3513,Z 162,A -102.0905,B 13.3995,C 0.1469,E1 13.3658,E2 192.0486} C_DIS
LIN {X -31.0474,Y -126.6323,Z 162,A -103.4722,B 13.3995,C 0.1458,E1 13.3621,E2 193.4288} C_DIS
LIN {X -34.1283,Y -125.8371,Z 162,A -104.8944,B 13.3995,C 0.1455,E1 13.3582,E2 194.8542} C_DIS
LIN {X -37.1897,Y -124.9667,Z 162,A -106.4584,B 13.3995,C 0.149,E1 13.354,E2 196.4378} C_DIS
LIN {X -41.78,Y -123.508,Z 162,A -108.4233,B 13.3995,C 0.1433,E1 13.3488,E2 198.3851} C_DIS
LIN {X -44.5666,Y -122.529,Z 162,A -109.7493,B 13.3995,C 0.1429,E1 13.3453,E2 199.7144} C_DIS
LIN {X -47.7812,Y -121.3123,Z 162,A -111.244,B 13.3995,C 0.1411,E1 13.3414,E2 201.2073} C_DIS
LIN {X -50.7391,Y -120.105,Z 162,A -112.6542,B 13.3995,C 0.1398,E1 13.3378,E2 202.6183} C_DIS
LIN {X -53.6666,Y -118.8255,Z 162,A -114.1984,B 13.3995,C 0.1419,E1 13.3338,E2 204.1789} C_DIS
LIN {X -57.8096,Y -116.865,Z 162,A -116.1213,B 13.3996,C 0.1372,E1 13.329,E2 206.0909} C_DIS
LIN {X -61.4678,Y -114.9855,Z 162,A -117.8953,B 13.3996,C 0.1341,E1 13.3246,E2 207.861} C_DIS
LIN {X -64.2667,Y -113.4453,Z 162,A -119.3116,B 13.3996,C 0.1325,E1 13.3211,E2 209.2785} C_DIS
LIN {X -67.0267,Y -111.8365,Z 162,A -120.8492,B 13.3996,C 0.134,E1 13.3174,E2 210.8316} C_DIS
LIN {X -70.5316,Y -109.6597,Z 162,A -122.5096,B 13.3997,C 0.1274,E1 13.3135,E2 212.4737} C_DIS
LIN {X -73.2152,Y -107.8863,Z 162,A -123.9691,B 13.3997,C 0.1264,E1 13.3101,E2 213.9382} C_DIS
LIN {X -76.3774,Y -105.6712,Z 162,A -125.6726,B 13.3997,C 0.1239,E1 13.3062,E2 215.642} C_DIS
LIN {X -79.2201,Y -103.557,Z 162,A -127.3396,B 13.3997,C 0.124,E1 13.3025,E2 217.3215} C_DIS
LIN {X -82.7555,Y -100.7547,Z 162,A -129.3047,B 13.3997,C 0.1201,E1 13.2982,E2 219.2838} C_DIS
LIN {X -85.7769,Y -98.1947,Z 162,A -131.0817,B 13.3997,C 0.1178,E1 13.2945,E2 221.0645} C_DIS
LIN {X -89.0579,Y -95.2295,Z 162,A -133.0212,B 13.3998,C 0.114,E1 13.2905,E2 223.0027} C_DIS
LIN {X -92.1935,Y -92.1977,Z 162,A -134.9894,B 13.3998,C 0.1115,E1 13.2865,E2 224.976} C_DIS
LIN {X -95.0132,Y -89.2885,Z 162,A -136.7653,B 13.3998,C 0.1077,E1 13.2831,E2 226.7505} C_DIS
LIN {X -97.9135,Y -86.0985,Z 162,A -138.6846,B 13.3999,C 0.1042,E1 13.2795,E2 228.6716} C_DIS
LIN {X -100.5693,Y -82.9804,Z 162,A -140.4642,B 13.3999,C 0.0998,E1 13.2764,E2 230.4479} C_DIS
LIN {X -103.0719,Y -79.8503,Z 162,A -142.253,B 13.3999,C 0.0965,E1 13.2733,E2 232.2388} C_DIS
LIN {X -105.1278,Y -77.1235,Z 162,A -143.7341,B 13.3999,C 0.0925,E1 13.2708,E2 233.7167} C_DIS
LIN {X -107.5149,Y -73.7592,Z 162,A -145.5208,B 13.4,C 0.0876,E1 13.2679,E2 235.4992} C_DIS
LIN {X -109.2887,Y -71.1047,Z 162,A -146.9344,B 13.4,C 0.0845,E1 13.2658,E2 236.913} C_DIS
LIN {X -110.9968,Y -68.4081,Z 162,A -148.4507,B 13.4,C 0.0838,E1 13.2635,E2 238.4414} C_DIS
LIN {X -113.1114,Y -64.852,Z 162,A -150.1859,B 13.4,C 0.0772,E1 13.2611,E2 240.1657} C_DIS
LIN {X -114.9887,Y -61.462,Z 162,A -152.0881,B 13.4,C 0.0777,E1 13.2585,E2 242.0897} C_DIS
LIN {X -116.8965,Y -57.7458,Z 162,A -153.7601,B 13.4001,C 0.0689,E1 13.2564,E2 243.7411} C_DIS
LIN {X -118.548,Y -54.2769,Z 162,A -155.6027,B 13.4001,C 0.0682,E1 13.2542,E2 245.6003} C_DIS
LIN {X -120.3482,Y -50.1567,Z 162,A -157.5095,B 13.4001,C 0.0612,E1 13.2521,E2 247.4972} C_DIS
LIN {X -121.646,Y -46.923,Z 162,A -159.0155,B 13.4001,C 0.0564,E1 13.2506,E2 248.999} C_DIS
LIN {X -122.7605,Y -43.9245,Z 162,A -160.5459,B 13.4001,C 0.0555,E1 13.2491,E2 250.5425} C_DIS
LIN {X -124.086,Y -40.0277,Z 162,A -162.4042,B 13.4002,C 0.0516,E1 13.2475,E2 252.4049} C_DIS
LIN {X -125.2245,Y -36.3093,Z 162,A -163.9898,B 13.4002,C 0.0439,E1 13.2462,E2 253.9746} C_DIS
LIN {X -126.0769,Y -33.2292,Z 162,A -165.4088,B 13.4002,C 0.0402,E1 13.2452,E2 255.3939} C_DIS
LIN {X -126.8537,Y -30.1293,Z 162,A -166.83,B 13.4002,C 0.0366,E1 13.2443,E2 256.8157} C_DIS
LIN {X -127.5601,Y -26.9844,Z 162,A -168.257,B 13.4002,C 0.0328,E1 13.2434,E2 258.2424} C_DIS
LIN {X -128.1827,Y -23.8551,Z 162,A -169.6721,B 13.4002,C 0.029,E1 13.2427,E2 259.6576} C_DIS
LIN {X -128.7286,Y -20.7117,Z 162,A -171.1093,B 13.4002,C 0.0258,E1 13.242,E2 261.0975} C_DIS
LIN {X -129.1077,Y -18.1864,Z 162,A -172.3497,B 13.4002,C 0.0253,E1 13.2415,E2 262.3502} C_DIS
LIN {X -129.661,Y -13.6958,Z 162,A -174.3018,B 13.4002,C 0.0185,E1 13.2409,E2 264.2959} C_DIS
LIN {X -129.9696,Y -10.3802,Z 162,A -175.7591,B 13.4002,C 0.0141,E1 13.2405,E2 265.7511} C_DIS
LIN {X -130.2142,Y -6.617,Z 162,A -177.4332,B 13.4002,C 0.0096,E1 13.2403,E2 267.4252} C_DIS
LIN {X -130.3556,Y -2.6863,Z 162,A -179.2751,B 13.4003,C 0.0071,E1 13.2401,E2 269.2782} C_DIS
LIN {X -130.3829,Y 0.4479,Z 162,A 179.3295,B 13.4003,C 0.0034,E1 13.2401,E2 270.6741} C_DIS
LIN {X -130.2938,Y 4.8087,Z 162,A 177.5101,B 13.4003,C -0.0046,E1 13.2402,E2 272.4801} C_DIS
LIN {X -130.1351,Y 8.0226,Z 162,A 176.0857,B 13.4003,C -0.0086,E1 13.2405,E2 273.9039} C_DIS
LIN {X -129.84,Y 11.8909,Z 162,A 174.2835,B 13.4003,C -0.0113,E1 13.2409,E2 275.7154} C_DIS
LIN {X -129.4817,Y 15.2965,Z 162,A 172.8349,B 13.4003,C -0.0171,E1 13.2413,E2 277.1557} C_DIS
LIN {X -129.1027,Y 18.2208,Z 162,A 171.4739,B 13.4003,C -0.0195,E1 13.2418,E2 278.5226} C_DIS
LIN {X -128.5787,Y 21.61,Z 162,A 170.0015,B 13.4003,C -0.0247,E1 13.2425,E2 279.9892} C_DIS
LIN {X -128.0076,Y 24.7707,Z 162,A 168.578,B 13.4003,C -0.0286,E1 13.2432,E2 281.4125} C_DIS
LIN {X -127.2137,Y 28.5717,Z 162,A 166.733,B 13.4003,C -0.0303,E1 13.2443,E2 283.2712} C_DIS
LIN {X -126.3082,Y 32.3379,Z 162,A 165.1045,B 13.4003,C -0.037,E1 13.2454,E2 284.8892} C_DIS
LIN {X -125.4137,Y 35.6531,Z 162,A 163.6022,B 13.4003,C -0.0416,E1 13.2465,E2 286.3889} C_DIS
LIN {X -124.3866,Y 39.0866,Z 162,A 161.9162,B 13.4003,C -0.0435,E1 13.2479,E2 288.0858} C_DIS
LIN {X -123.2902,Y 42.4149,Z 162,A 160.4449,B 13.4003,C -0.0495,E1 13.2492,E2 289.5472} C_DIS
LIN {X -121.8813,Y 46.3111,Z 162,A 158.629,B 13.4002,C -0.0548,E1 13.251,E2 291.3604} C_DIS
LIN {X -120.7118,Y 49.2785,Z 162,A 157.1885,B 13.4002,C -0.0578,E1 13.2525,E2 292.8035} C_DIS
LIN {X -119.4695,Y 52.2177,Z 162,A 155.7707,B 13.4002,C -0.0613,E1 13.254,E2 294.2214} C_DIS
LIN {X -118.1552,Y 55.1264,Z 162,A 154.2313,B 13.4002,C -0.0619,E1 13.2558,E2 295.7747} C_DIS
LIN {X -116.4666,Y 58.6112,Z 162,A 152.6456,B 13.4002,C -0.0693,E1 13.2578,E2 297.345} C_DIS
LIN {X -114.7438,Y 61.9177,Z 162,A 150.8722,B 13.4002,C -0.0704,E1 13.2601,E2 299.1319} C_DIS
LIN {X -112.6385,Y 65.6706,Z 162,A 149.0658,B 13.4001,C -0.0774,E1 13.2626,E2 300.9263} C_DIS
LIN {X -110.999,Y 68.4045,Z 162,A 147.6526,B 13.4001,C -0.0808,E1 13.2646,E2 302.3392} C_DIS
LIN {X -108.9223,Y 71.6646,Z 162,A 145.8917,B 13.4001,C -0.0836,E1 13.2673,E2 304.1052} C_DIS
LIN {X -106.599,Y 75.077,Z 162,A 144.111,B 13.4001,C -0.0889,E1 13.2701,E2 305.8798} C_DIS
LIN {X -104.3226,Y 78.2102,Z 162,A 142.2823,B 13.4001,C -0.0901,E1 13.2732,E2 307.721} C_DIS
LIN {X -101.7882,Y 81.4811,Z 162,A 140.4792,B 13.4,C -0.0948,E1 13.2763,E2 309.5202} C_DIS
LIN {X -99.2459,Y 84.5586,Z 162,A 138.7015,B 13.4,C -0.0983,E1 13.2795,E2 311.2985} C_DIS
LIN {X -96.6101,Y 87.5579,Z 162,A 136.931,B 13.4,C -0.1019,E1 13.2828,E2 313.0688} C_DIS
LIN {X -93.8845,Y 90.4747,Z 162,A 135.0939,B 13.4,C -0.1038,E1 13.2863,E2 314.9133} C_DIS
LIN {X -90.7223,Y 93.6448,Z 162,A 133.1975,B 13.3999,C -0.1098,E1 13.2901,E2 316.7993} C_DIS
LIN {X -87.8133,Y 96.3783,Z 162,A 131.3599,B 13.3999,C -0.1114,E1 13.2939,E2 318.6445} C_DIS
LIN {X -84.5635,Y 99.2417,Z 162,A 129.482,B 13.3999,C -0.1159,E1 13.2978,E2 320.5173} C_DIS
LIN {X -81.4668,Y 101.7996,Z 162,A 127.6924,B 13.3998,C -0.1187,E1 13.3017,E2 322.3079} C_DIS
LIN {X -78.2146,Y 104.3193,Z 162,A 125.9919,B 13.3998,C -0.1247,E1 13.3054,E2 323.9942} C_DIS
LIN {X -75.6092,Y 106.2225,Z 162,A 124.4537,B 13.3998,C -0.1243,E1 13.3089,E2 325.5446} C_DIS
LIN {X -72.4396,Y 108.4085,Z 162,A 122.7617,B 13.3998,C -0.1273,E1 13.3128,E2 327.2349} C_DIS
LIN {X -68.9758,Y 110.6447,Z 162,A 120.9077,B 13.3997,C -0.1292,E1 13.3172,E2 329.0918} C_DIS
LIN {X -65.2757,Y 112.8671,Z 162,A 119.009,B 13.3997,C -0.1322,E1 13.3218,E2 330.9889} C_DIS
LIN {X -61.4354,Y 115.003,Z 162,A 116.9888,B 13.3997,C -0.1329,E1 13.3268,E2 333.0174} C_DIS
LIN {X -57.7884,Y 116.8755,Z 162,A 115.2958,B 13.3997,C -0.1381,E1 13.3309,E2 334.6962} C_DIS
LIN {X -54.3006,Y 118.5371,Z 162,A 113.6706,B 13.3996,C -0.1422,E1 13.335,E2 336.3117} C_DIS
Enddeposition()
END
